# B&R Automation Studio project CombinedLinenCleanA6 (part 3)

#### 6_sdc1.var
```iecst
VAR RETAIN
	STEP : UINT;
	PLS : BOOL;
	LASTSTEP : UINT;
	SteadyUp : BOOL;
	CloserUpET : TIME;
	SteadysDown : BOOL;
	SteadysDownET : TIME;
	LoadDropped : BOOL;
END_VAR
VAR
	SteadyUpET : TIME;
	CloserDownET : TIME;
	SettledAtDischargerET : TIME;
	MinOpenET : TIME;
	SettledAtDischarger : BOOL;
	CloserDown : BOOL;
	MinOpen : BOOL;
	CloserUp : BOOL;
	SettledAtBuffer : BOOL;
	SettledAtBufferET : TIME;
	I_BagAtBuffer : BOOL;
	O_OpenStop : BOOL;
	O_OpenBag : BOOL;
	O_Steadys : BOOL;
	O_OpenBuffer : BOOL;
	O_Closer : BOOL;
	I_BagAtDischarger : BOOL;
	I_OpenBag : BOOL;
	I_LoadDropped : BOOL;
	TestDrop : BOOL;
	DischargerEnable : BOOL;
	TestDischarger : BOOL;
	Remainder : SINT;
	TimerAlarm : TON_10ms;
	WgtRound : UINT;
	a : BOOL;
	I_BagEmpty : BOOL;
	MySeq : USINT;
	O_BagReady : BOOL;
	O_JoinCDC4 : BOOL;
END_VAR
```

#### 6_sdc1Cyclic.ab
```automation-basic
PROGRAM _CYCLIC
	(* cyclic program *)

;Sequence 6 - Discharger 1 D[906]
a

;-----------------------------------------
;Revision 1.00 19/12/2005 D.J. First Issue
;-----------------------------------------

DischargerEnable 		= ((D[24] > 0) AND NOT Std.HaltSys)
MySeq                       = 9

//I_BagAtBuffer			  = X[3].X08
I_BagAtDischarger = X[3].X11
//I_SafetyRunning       = X[8].X15

I_OpenBag				= Enable.CDC4Open OR TestDrop           ;X[23].X01
//I_LoadDropped			= X[7].X13 OR TestDischarger  ;X[23].X02
//I_BagEmpty              = X[2].X13

O_Steadys				= FALSE ;Y[6].Y01
O_OpenBuffer 			= FALSE ;Y[6].Y02
O_OpenBag				= FALSE ;Y[6].Y03
O_OpenStop				= FALSE ;Y[6].Y04
O_Closer				= FALSE ;Y[6].Y05
O_BagReady          = FALSE
O_JoinCDC4           = FALSE
Request.CDC[4] 	     = FALSE

;Alarm
Alarm[MySeq].Name 			= 0 ;Clear sequence alarm name
Alarm[MySeq].Bag 			= 45
Alarm[MySeq].Beacon			= TRUE
Alarm[MySeq].Extra			= 0
Alarm[MySeq].Time			= 3000

;Setup Sequence
STEP = D[900+MySeq]
;Setup Pulse contact
PLS = (STEP <> LASTSTEP)
LASTSTEP = STEP

;Step 0 - Disabled
IF (STEP = 0) THEN
	;Disabled
ENDIF

;Check Status - Bag settled at buffer, no bag at discharger, bag at buffer on screen and no bag at discharger on the screen
TON_10ms(I_BagAtBuffer,300,SettledAtBuffer,SettledAtBufferET)
IF (STEP = 1) THEN
	IF DischargerEnable AND   NOT I_BagAtDischarger AND (Bag[45].Cat = 0) THEN
		D[900+MySeq] = 2
	ENDIF
	IF (Bag[45].Cat > 0) THEN
		Alarm[MySeq].Name = almBagDataError
	ELSE IF I_BagAtDischarger THEN
		Alarm[MySeq].Name = almSwitchFault
	ENDIF
ENDIF

;Wait for bag in discharger
IF (STEP = 2) THEN
	Request.CDC[4] 	= TRUE
;	IF (Bag[44].Cat = 0) AND (Bag[11].Cat>0) THEN
;		Bag[44] = Bag[11]
;		Bag[11]   = Bag[0]
;	ENDIF
	IF I_BagAtDischarger THEN
		D[900+MySeq] = 3
	ENDIF
	Alarm[7].Name = almBagNotArrived
ENDIF

;Let bag settle in discharger
TON_10ms(((STEP = 3) AND I_BagAtDischarger),1000,SettledAtDischarger,SettledAtDischargerET)
IF (STEP = 3) THEN
;	IF (Bag[228].Cat = 0) AND (Bag[227].Cat > 0) THEN
;		Bag[228] = Bag[227]
;		Bag[227] = Bag[0]
;	ENDIF
	IF SettledAtDischarger THEN
		D[900+MySeq] = 4
	ENDIF
	Alarm[MySeq].Name = almBagNotSettled
ENDIF

;Allow steadys to move down
TON_10ms((STEP = 4),400,SteadysDown,SteadysDownET)
IF (STEP = 4) THEN
	IF SteadysDown AND (Bag[45].Cat <> Std.MaxCats)  THEN
		D[900+MySeq] = 5
	ENDIF
	IF (Bag[45].Cat = Std.MaxCats) AND SteadysDown THEN
		D[900+MySeq] = 8
	ENDIF
ENDIF

;Steady cylinders on from steps 4 - 9
O_Steadys = ((STEP >= 4) AND (STEP <= 9))

;Bag opener on from step 5 - 8
O_OpenBag = ((STEP >= 6) AND (STEP <= 8))

;Wash Codes
;IF (STEP = 4) OR (STEP = 5) THEN
;
;;round up weight to give to wash machine
;	Remainder = SINT(Bag[228].Wgt MOD 10)
;	IF (Remainder > 4) THEN
;		WgtRound = (Bag[228].Wgt + 10)
;	ELSE
;		WgtRound = Bag[228].Wgt
;	ENDIF
;
;
;;Codes to CBW
;	CAN[1].Category = Bag[228].Cat
;	CAN[1].Customer = Bag[228].Cus
;	CAN[1].Weight   = (WgtRound / 10)
;ELSE
;	CAN[1].Category = 0
;	CAN[1].Customer = 0
;	CAN[1].Weight   = 0
;ENDIF

;Bag Ready to Washing Machine
IF (STEP = 5) THEN
	O_BagReady = TRUE
	O_Closer        = TRUE  ;  ????????????????????????
	IF I_OpenBag OR TestDischarger THEN
		D[900+MySeq] = 6
	ENDIF

ENDIF

;Open Bag Until LoadDropped recieved and has been open for 6 seconds
TON_10ms((STEP = 6),600,MinOpen,MinOpenET) ;ET means Elapsed Time
IF (STEP = 6) THEN
	IF  I_OpenBag THEN
		LoadDropped = TRUE
	ENDIF
	IF (NOT I_OpenBag AND MinOpen) THEN
		D[900+MySeq] = 7
	ENDIF
	Alarm[MySeq].Name = almLoadNotDropped
	ELSE
	LoadDropped = FALSE
ENDIF

;Change display to empty bag
IF (STEP = 7) THEN
	O_BagReady = Std.Clock500ms
	IF (D[927]>3) THEN
		LoadDropped = TRUE
	ENDIF
	IF (LoadDropped  OR TestDrop) THEN ;AND I_BagEmpty) OR TestDrop) THEN
		Bag[45].Cat 	= Std.MaxCats
		D[900+MySeq] 			= 8
	ENDIF
	Alarm[MySeq].Name = almGeneralSequence
	ELSE
	LoadDropped = FALSE
ENDIF

;Close bag
TON_10ms((STEP = 8),700,CloserDown,CloserDownET)
IF (STEP = 8) THEN
	O_Closer = TRUE
	IF CloserDown THEN
		D[900+MySeq] = 9
	ENDIF
ENDIF

;Allow closer to go back up
TON_10ms((STEP = 9),700,CloserUp,CloserUpET)
IF (STEP = 9) THEN
	IF CloserUp THEN
		D[900+MySeq] = 10
	ENDIF
ENDIF

;Allow steadys to go up
TON_10ms((STEP = 10),400,SteadyUp,SteadyUpET)
IF (STEP = 10) THEN
	IF SteadyUp THEN
		D[900+MySeq] = 11
	ENDIF
ENDIF

;Check for space on empty bag buffer
IF (STEP = 11) THEN
 	Request.CDC4Empty = TRUE
	IF Enable.CDC4Empty  THEN
		D[900+MySeq] = 12
	ENDIF
	ELSE
		Request.CDC4Empty = FALSE
ENDIF

;Open buffer stop - unitl bag out
IF (STEP = 12) THEN
	O_OpenStop = TRUE
	O_JoinCDC4 = TRUE
	IF PLS THEN
		Bag[42].Cat = 99
	ENDIF
	Bag[45].Cat = 0
	Bag[45].Cus = 0
	Bag[45].Wgt = 0
	IF NOT Enable.CDC4Empty AND NOT I_BagAtDischarger THEN
		D[900+MySeq] = 1
	ENDIF
	Alarm[MySeq].Name = almBagNotReleased
ENDIF

;Alarms
TimerAlarm.IN 	= NOT PLS AND (Alarm[MySeq].Name > 0)
TimerAlarm.PT 	= Alarm[MySeq].Time
TimerAlarm FUB TON_10ms()
Alarm[MySeq].On 	= TimerAlarm.Q
Alarm[MySeq].ET 	= TimerAlarm.ET

;Outputs

//Y[3].Y10 = O_OpenBuffer
Y[3].Y16 = O_Steadys
Y[4].Y01 = O_OpenBag
Y[4].Y02 = O_OpenStop
Y[4].Y03 = O_Closer
Y[7].Y01= O_JoinCDC4
END_PROGRAM
```

### Program Logical/Sequences/10ms/10_sdc5 (IEC, version 1.00.0) - * SDC1 Machine 1 BCD/CAN

#### 6_sdc1Cyclic.ab
```automation-basic
PROGRAM _CYCLIC
	(* cyclic program *)

;Sequence 6 - Discharger 1 D[906]
a

;-----------------------------------------
;Revision 1.00 19/12/2005 D.J. First Issue
;-----------------------------------------

DischargerEnable 		= ((D[25] > 0) AND NOT Std.HaltSys)
MySeq                       = 10

I_BagAtBuffer			  = X[3].X15
I_BagAtDischarger = X[3].X14
//I_SafetyRunning       = X[8].X15

I_OpenBag				= X[4].X01 OR TestDrop           ;X[23].X01
//I_LoadDropped			= X[7].X13 OR TestDischarger  ;X[23].X02
//I_BagEmpty              = X[2].X13

O_Steadys				= FALSE ;Y[6].Y01
O_OpenBuffer 			= FALSE ;Y[6].Y02
O_OpenBag				= FALSE ;Y[6].Y03
O_OpenStop				= FALSE ;Y[6].Y04
O_Closer				= FALSE ;Y[6].Y05
O_BagReady          = FALSE
Request.CDC[6]     = FALSE

;Alarm
Alarm[MySeq].Name 			= 0 ;Clear sequence alarm name
Alarm[MySeq].Bag 			= 46
Alarm[MySeq].Beacon			= TRUE
Alarm[MySeq].Extra			= 0
Alarm[MySeq].Time			= 3000

;Setup Sequence
STEP = D[900+MySeq]
;Setup Pulse contact
PLS = (STEP <> LASTSTEP)
LASTSTEP = STEP

;Step 0 - Disabled
IF (STEP = 0) THEN
	;Disabled
ENDIF

;Check Status - Bag settled at buffer, no bag at discharger, bag at buffer on screen and no bag at discharger on the screen
TON_10ms(I_BagAtBuffer,300,SettledAtBuffer,SettledAtBufferET)
IF (STEP = 1) THEN
	IF DischargerEnable AND SettledAtBuffer AND  NOT I_BagAtDischarger AND (Bag[46].Cat = 0) AND (Bag[26].Cat > 0)THEN
		D[900+MySeq] = 2
	ENDIF
	IF (Bag[46].Cat > 0) THEN
		Alarm[MySeq].Name = almBagDataError
	ELSE IF I_BagAtDischarger THEN
		Alarm[MySeq].Name = almSwitchFault
	ENDIF
ENDIF

;Wait for bag in discharger
IF (STEP = 2) THEN
	O_OpenBuffer 	= TRUE

	IF I_BagAtDischarger THEN
		D[900+MySeq] = 3
	ENDIF
	Alarm[7].Name = almBagNotArrived
ENDIF

;Let bag settle in discharger
TON_10ms(((STEP = 3) AND I_BagAtDischarger),1000,SettledAtDischarger,SettledAtDischargerET)
IF (STEP = 3) THEN
	IF (Bag[46].Cat = 0) AND (Bag[26].Cat>0) THEN
		Bag[46] = Bag[26]
		Bag[26]   = Bag[0]
	ENDIF
	IF SettledAtDischarger THEN
		D[900+MySeq] = 4
	ENDIF
	Alarm[MySeq].Name = almBagNotSettled
ENDIF

;Allow steadys to move down
TON_10ms((STEP = 4),400,SteadysDown,SteadysDownET)
IF (STEP = 4) THEN
	IF SteadysDown AND (Bag[46].Cat <> Std.MaxCats)  THEN
		D[900+MySeq] = 5
	ENDIF
	IF (Bag[46].Cat = Std.MaxCats) AND SteadysDown THEN
		D[900+MySeq] = 8
	ENDIF
ENDIF

;Steady cylinders on from steps 4 - 9
O_Steadys = ((STEP >= 4) AND (STEP <= 9))

;Bag opener on from step 5 - 8
O_OpenBag = ((STEP >= 6) AND (STEP <= 8))

;Wash Codes
;IF (STEP = 4) OR (STEP = 5) THEN
;
;;round up weight to give to wash machine
;	Remainder = SINT(Bag[228].Wgt MOD 10)
;	IF (Remainder > 4) THEN
;		WgtRound = (Bag[228].Wgt + 10)
;	ELSE
;		WgtRound = Bag[228].Wgt
;	ENDIF
;
;
;;Codes to CBW
;	CAN[1].Category = Bag[228].Cat
;	CAN[1].Customer = Bag[228].Cus
;	CAN[1].Weight   = (WgtRound / 10)
;ELSE
;	CAN[1].Category = 0
;	CAN[1].Customer = 0
;	CAN[1].Weight   = 0
;ENDIF

;Bag Ready to Washing Machine
IF (STEP = 5) THEN
	O_BagReady = TRUE
	O_Closer        = TRUE
	IF I_OpenBag OR TestDischarger THEN
		D[900+MySeq] = 6
	ENDIF

ENDIF

;Open Bag Until LoadDropped recieved and has been open for 6 seconds
TON_10ms((STEP = 6),600,MinOpen,MinOpenET) ;ET means Elapsed Time
IF (STEP = 6) THEN
	IF I_OpenBag THEN
		LoadDropped = TRUE
	ENDIF
	IF (NOT I_OpenBag AND MinOpen) THEN
		D[900+MySeq] = 7
	ENDIF
	Alarm[MySeq].Name = almLoadNotDropped
	ELSE
	LoadDropped = FALSE
ENDIF

;Change display to empty bag
IF (STEP = 7) THEN
	O_BagReady = TRUE
	IF I_OpenBag THEN
		LoadDropped = TRUE
	ENDIF
	IF (LoadDropped  OR TestDrop) THEN ;AND I_BagEmpty) OR TestDrop) THEN
		Bag[46].Cat 	= Std.MaxCats
		D[900+MySeq] 			= 8
	ENDIF
	Alarm[MySeq].Name = almGeneralSequence
	ELSE
	LoadDropped = FALSE
ENDIF

;Close bag
TON_10ms((STEP = 8),700,CloserDown,CloserDownET)
IF (STEP = 8) THEN
	O_Closer = TRUE
	IF CloserDown THEN
		D[900+MySeq] = 9
	ENDIF
ENDIF

;Allow closer to go back up
TON_10ms((STEP = 9),700,CloserUp,CloserUpET)
IF (STEP = 9) THEN
	IF CloserUp THEN
		D[900+MySeq] = 10
	ENDIF
ENDIF

;Allow steadys to go up
TON_10ms((STEP = 10),400,SteadyUp,SteadyUpET)
IF (STEP = 10) THEN
	IF SteadyUp THEN
		D[900+MySeq] = 11
	ENDIF
ENDIF

;Check for space on empty bag buffer
IF (STEP = 11) THEN
 	Request.CDC[5] = TRUE
	IF Enable.CDC[5]  THEN
		D[900+MySeq] = 12
	ENDIF
	ELSE
		Request.CDC[5] = FALSE
ENDIF

;Open buffer stop - unitl bag out
IF (STEP = 12) THEN
	O_OpenStop = TRUE
	IF PLS THEN
		;C[14] = 0
	ENDIF
	Bag[46].Cat = 0
	Bag[46].Cus = 0
	Bag[46].Wgt = 0
	IF NOT Enable.CDC[5]  THEN
		D[900+MySeq] = 1
	ENDIF
	Alarm[MySeq].Name = almBagNotReleased
ENDIF

;Alarms
TimerAlarm.IN 	= NOT PLS AND (Alarm[MySeq].Name > 0)
TimerAlarm.PT 	= Alarm[MySeq].Time
TimerAlarm FUB TON_10ms()
Alarm[MySeq].On 	= TimerAlarm.Q
Alarm[MySeq].ET 	= TimerAlarm.ET

;Outputs

Y[4].Y06 = O_OpenBuffer
Y[4].Y07 = O_Steadys
Y[4].Y08 = O_OpenBag
Y[4].Y09 = O_OpenStop
Y[4].Y10 = O_Closer

END_PROGRAM
```

#### 6_sdc1.var
```iecst
VAR RETAIN
	STEP : UINT;
	PLS : BOOL;
	LASTSTEP : UINT;
	SteadyUp : BOOL;
	CloserUpET : TIME;
	SteadysDown : BOOL;
	SteadysDownET : TIME;
	LoadDropped : BOOL;
END_VAR
VAR
	SteadyUpET : TIME;
	CloserDownET : TIME;
	SettledAtDischargerET : TIME;
	MinOpenET : TIME;
	SettledAtDischarger : BOOL;
	CloserDown : BOOL;
	MinOpen : BOOL;
	CloserUp : BOOL;
	SettledAtBuffer : BOOL;
	SettledAtBufferET : TIME;
	I_BagAtBuffer : BOOL;
	O_OpenStop : BOOL;
	O_OpenBag : BOOL;
	O_Steadys : BOOL;
	O_OpenBuffer : BOOL;
	O_Closer : BOOL;
	I_BagAtDischarger : BOOL;
	I_OpenBag : BOOL;
	I_LoadDropped : BOOL;
	TestDrop : BOOL;
	DischargerEnable : BOOL;
	TestDischarger : BOOL;
	Remainder : SINT;
	TimerAlarm : TON_10ms;
	WgtRound : UINT;
	a : BOOL;
	I_BagEmpty : BOOL;
	MySeq : USINT;
	O_BagReady : BOOL;
END_VAR
```

### Program Logical/Sequences/10ms/11_sdc6 (IEC) - * SDC1 Machine 1 BCD/CAN

#### 6_sdc1Cyclic.ab
```automation-basic
PROGRAM _CYCLIC
	(* cyclic program *)

;Sequence 6 - Discharger 1 D[906]
a

;-----------------------------------------
;Revision 1.00 19/12/2005 D.J. First Issue
;-----------------------------------------

DischargerEnable 		= ((D[26] > 0) AND NOT Std.HaltSys)
MySeq                       = 11

I_BagAtBuffer			  = X[6].X08
I_BagAtDischarger = X[4].X02
//I_SafetyRunning       = X[8].X15

I_OpenBag				= X[4].X04 OR TestDrop           ;X[23].X01
//I_LoadDropped			= X[7].X13 OR TestDischarger  ;X[23].X02
//I_BagEmpty              = X[2].X13

O_Steadys				= FALSE ;Y[6].Y01
O_OpenBuffer 			= FALSE ;Y[6].Y02
O_OpenBag				= FALSE ;Y[6].Y03
O_OpenStop				= FALSE ;Y[6].Y04
O_Closer				= FALSE ;Y[6].Y05
O_BagReady          = FALSE

;Alarm
Alarm[MySeq].Name 			= 0 ;Clear sequence alarm name
Alarm[MySeq].Bag 			= 47
Alarm[MySeq].Beacon			= TRUE
Alarm[MySeq].Extra			= 0
Alarm[MySeq].Time			= 3000

;Setup Sequence
STEP = D[900+MySeq]
;Setup Pulse contact
PLS = (STEP <> LASTSTEP)
LASTSTEP = STEP

;Step 0 - Disabled
IF (STEP = 0) THEN
	;Disabled
ENDIF

;Check Status - Bag settled at buffer, no bag at discharger, bag at buffer on screen and no bag at discharger on the screen
TON_10ms(I_BagAtBuffer,300,SettledAtBuffer,SettledAtBufferET)
IF (STEP = 1) THEN
	IF DischargerEnable AND SettledAtBuffer AND  NOT I_BagAtDischarger AND (Bag[47].Cat = 0) AND (Bag[21].Cat > 0)THEN
		D[900+MySeq] = 2
	ENDIF
	IF (Bag[47].Cat > 0) THEN
		Alarm[MySeq].Name = almBagDataError
	ELSE IF I_BagAtDischarger THEN
		Alarm[MySeq].Name = almSwitchFault
	ENDIF
ENDIF

;Wait for bag in discharger
IF (STEP = 2) THEN
	O_OpenBuffer 	= TRUE

	IF I_BagAtDischarger THEN
		D[900+MySeq] = 3
	ENDIF
	Alarm[7].Name = almBagNotArrived
ENDIF

;Let bag settle in discharger
TON_10ms(((STEP = 3) AND I_BagAtDischarger),1000,SettledAtDischarger,SettledAtDischargerET)
IF (STEP = 3) THEN
	IF (Bag[47].Cat = 0) AND (Bag[21].Cat>0) THEN
		Bag[47] = Bag[21]
		Bag[21]   = Bag[0]
	ENDIF
	IF SettledAtDischarger THEN
		D[900+MySeq] = 4
	ENDIF
	Alarm[MySeq].Name = almBagNotSettled
ENDIF

;Allow steadys to move down
TON_10ms((STEP = 4),400,SteadysDown,SteadysDownET)
IF (STEP = 4) THEN
	IF SteadysDown AND (Bag[47].Cat <> Std.MaxCats)  THEN
		D[900+MySeq] = 5
	ENDIF
	IF (Bag[47].Cat = Std.MaxCats) AND SteadysDown THEN
		D[900+MySeq] = 8
	ENDIF
ENDIF

;Steady cylinders on from steps 4 - 9
O_Steadys = ((STEP >= 4) AND (STEP <= 9))

;Bag opener on from step 5 - 8
O_OpenBag = ((STEP >= 6) AND (STEP <= 8))

;Wash Codes
;IF (STEP = 4) OR (STEP = 5) THEN
;
;;round up weight to give to wash machine
;	Remainder = SINT(Bag[228].Wgt MOD 10)
;	IF (Remainder > 4) THEN
;		WgtRound = (Bag[228].Wgt + 10)
;	ELSE
;		WgtRound = Bag[228].Wgt
;	ENDIF
;
;
;;Codes to CBW
;	CAN[1].Category = Bag[228].Cat
;	CAN[1].Customer = Bag[228].Cus
;	CAN[1].Weight   = (WgtRound / 10)
;ELSE
;	CAN[1].Category = 0
;	CAN[1].Customer = 0
;	CAN[1].Weight   = 0
;ENDIF

;Bag Ready to Washing Machine
IF (STEP = 5) THEN
	O_BagReady = TRUE
	O_Closer        = TRUE
	IF I_OpenBag OR TestDischarger THEN
		D[900+MySeq] = 6
	ENDIF

ENDIF

;Open Bag Until LoadDropped recieved and has been open for 6 seconds
TON_10ms((STEP = 6),600,MinOpen,MinOpenET) ;ET means Elapsed Time
IF (STEP = 6) THEN
	IF I_OpenBag THEN
//		LoadDropped = TRUE
	ENDIF
	IF (NOT I_OpenBag AND MinOpen) THEN
		D[900+MySeq] = 7
	ENDIF
;	Alarm[MySeq].Name = almLoadNotDropped
	ELSE
//	LoadDropped = FALSE
ENDIF

;Change display to empty bag
IF (STEP = 7) THEN
	O_BagReady = TRUE
	IF I_OpenBag THEN
		LoadDropped = TRUE
	ENDIF
	IF (LoadDropped  OR TestDrop) THEN ;AND I_BagEmpty) OR TestDrop) THEN
		Bag[47].Cat 	= Std.MaxCats
		D[900+MySeq] 			= 8
	ENDIF
	;Alarm[MySeq].Name = almGeneralSequence
	ELSE
	LoadDropped = FALSE
ENDIF

;Close bag
TON_10ms((STEP = 8),700,CloserDown,CloserDownET)
IF (STEP = 8) THEN
	O_Closer = TRUE
	IF CloserDown THEN
		D[900+MySeq] = 9
	ENDIF
ENDIF

;Allow closer to go back up
TON_10ms((STEP = 9),700,CloserUp,CloserUpET)
IF (STEP = 9) THEN
	IF CloserUp THEN
		D[900+MySeq] = 10
	ENDIF
ENDIF

;Allow steadys to go up
TON_10ms((STEP = 10),400,SteadyUp,SteadyUpET)
IF (STEP = 10) THEN
	IF SteadyUp THEN
		D[900+MySeq] = 11
	ENDIF
ENDIF

;Check for space on empty bag buffer
IF (STEP = 11) THEN
 	Request.CDC[6] = TRUE
	IF Enable.CDC[6]  THEN
		D[900+MySeq] = 12
	ENDIF
	ELSE
		Request.CDC[6] = FALSE
ENDIF

;Open buffer stop - unitl bag out
IF (STEP = 12) THEN
	O_OpenStop = TRUE
	IF PLS THEN
		;C[14] = 0
	ENDIF
	Bag[47].Cat = 0
	Bag[47].Cus = 0
	Bag[47].Wgt = 0
	IF NOT Enable.CDC[6]  THEN
		D[900+MySeq] = 1
	ENDIF
	Alarm[MySeq].Name = almBagNotReleased
ENDIF

;Alarms
TimerAlarm.IN 	= NOT PLS AND (Alarm[MySeq].Name > 0)
TimerAlarm.PT 	= Alarm[MySeq].Time
TimerAlarm FUB TON_10ms()
Alarm[MySeq].On 	= TimerAlarm.Q
Alarm[MySeq].ET 	= TimerAlarm.ET

;Outputs

Y[4].Y16 = O_BagReady
Y[8].Y16 = O_OpenBuffer
Y[4].Y12 = O_Steadys
Y[4].Y13 = O_OpenBag
Y[4].Y14 = O_OpenStop
Y[4].Y15 = O_Closer

END_PROGRAM
```

### Program Logical/Sequences/10ms/12_ebag (IEC) - *PUP1 Unloading point

#### pup.var
```iecst
VAR RETAIN
	LASTSTEP : UINT;
	PLS : BOOL;
	STEP : UINT;
END_VAR
VAR
	TimerAlarm : TON_10ms;
	mySeq : UINT;
	myIO : UINT;
	I_ReleasePB : BOOL;
	I_UnloadingPointOn : BOOL;
	I_TrolleyReleased : BOOL;
	I_BagAtBuffer : BOOL;
	I_BagReleasedBuffer : BOOL;
	myBag : UINT;
	O_Lamp : BOOL;
	O_OpenBuffer : BOOL;
	O_Release : BOOL;
	myPup : UINT;
	SettledBuffer : BOOL;
	SettledBufferET : UDINT;
	myBufferBag : UINT;
	BagReleased : BOOL;
	myZone : INT;
	I_BagInSep : BOOL;
	SettledInSep : BOOL;
	SettledInSepET : UDINT;
	O_SelectCDC3 : BOOL;
	O_SelectCIC3 : BOOL;
END_VAR
```

#### pup.ab
```automation-basic
;--------------------------------------------
;Sequence 0 - XXX0  D[900 + mySeq]
;--------------------------------------------

PROGRAM _INIT
(* init program *)
END_PROGRAM

PROGRAM _CYCLIC

;Inputs
mySeq				= 12	;Sequence number
//myIO				= 345
//myBu/fferBag			= 950
//myBa/g				= 987
//myPup				= 1
//myZone				= 0

I_BagAtBuffer		= X[myIO].X01
I_BagInSep			= X[myIO].X02
I_UnloadingPointOn	= X[myIO].X03
I_ReleasePB			= X[myIO].X04
I_TrolleyReleased	= X[myIO].X08 ; Also Line full

Enable.CDC[3]  = FALSE
Enable.CIC[3]    = FALSE

//PUP[myPup].WorkingLamp = FALSE
O_SelectCIC3        = FALSE
O_SelectCDC3       = FALSE

Alarm[mySeq].Name 	= 0
Alarm[mySeq].Bag	= myBag
Alarm[mySeq].Beacon	= TRUE
Alarm[mySeq].Extra	= 0
Alarm[mySeq].Time	= 3000

;Setup Sequence
STEP = D[900 + mySeq]
;Setup Pulse contact
PLS = (STEP <> LASTSTEP)
LASTSTEP = STEP

;Sequence
IF (STEP = 0) THEN
	;Disabled
ENDIF

;Step 1 Wiat for bag at buffer.
TON_10ms(I_BagAtBuffer,75,SettledBuffer,SettledBufferET)
IF (STEP = 1) THEN
	IF Line[9].Clear THEN
		D[900 + mySeq] = 2
	ENDIF
	//	Alarm[mySeq].Name = almBagDataError

ENDIF

;Step 2 Release bag from Buffer
//TON_10ms(I_BagInSep,150,SettledInSep,SettledInSepET)
IF (STEP = 2) THEN
	IF Request.CDC[3] THEN
		C[9] = 0
		D[900 + mySeq] = 3
	ELSE IF Request.CIC[3] THEN
		C[9] = 0
		D[900 + mySeq] = 4
	ENDIF
	//	Alarm[mySeq].Bag = myBufferBag
	//	Alarm[mySeq].Name = almBagNotReleased

ENDIF

;Step 3 wait for pushbutton to request release of trolley
IF (STEP = 3) THEN
	O_SelectCDC3 = TRUE
	Enable.CDC[3] = TRUE
	IF Line[9].Trip THEN
		D[900 + mySeq] = 1
	ENDIF
		Alarm[mySeq].Name = almBagNotArrived
ENDIF

;STEP 4 Check for space in empty trolley buffer.
IF (STEP = 4) THEN
	O_SelectCIC3 = TRUE
	Enable.CIC[3]  = TRUE
	IF Line[9].Trip THEN
		D[900 + mySeq] = 1
	ENDIF
		Alarm[mySeq].Name = almBagNotArrived
ENDIF

;-----------------------------------
;PLC Outputs - adjust to suit system
;-----------------------------------

Y[6].Y10 = O_SelectCIC3
Y[6].Y09 = O_SelectCDC3

;Alarms
TimerAlarm.IN 		= NOT PLS AND (Alarm[mySeq].Name > 0)
TimerAlarm.PT 		= Alarm[mySeq].Time
TimerAlarm FUB TON_10ms()
Alarm[mySeq].On 	= TimerAlarm.Q
Alarm[mySeq].ET 	= TimerAlarm.ET
//Alarm[mySeq].Zone 	= myZone
END_PROGRAM
```

### Program Logical/Sequences/10ms/13_fb_eb (IEC) - *PUP5 Unloading point

#### pup.var
```iecst
VAR RETAIN
	LASTSTEP : UINT;
	PLS : BOOL;
	STEP : UINT;
END_VAR
VAR
	TimerAlarm : TON_10ms;
	mySeq : UINT;
	myIO : UINT;
	I_ReleasePB : BOOL;
	I_UnloadingPointOn : BOOL;
	I_TrolleyReleased : BOOL;
	myBag : UINT;
	O_Lamp : BOOL;
	O_OpenBuffer : BOOL;
	O_Release : BOOL;
	myPup : UINT;
	SettledBuffer : BOOL;
	SettledBufferET : UDINT;
	PUPValid : BOOL;
	myZone : INT;
	I_BagAtEmpty : BOOL;
	I_BagAtLine1 : BOOL;
	I_BagAtLine2 : BOOL;
	I_CDC1PB : BOOL;
	I_CDC1SelectLine1 : BOOL;
	I_CDC1SelectLine4 : BOOL;
	I_CDC4PB : BOOL;
	I_CDC4SelectLine1 : BOOL;
	I_CDC4SelectLine4 : BOOL;
	O_ResetPoints : BOOL;
	O_OpenEmpty : BOOL;
	O_OpenLine1 : BOOL;
	O_OpenLine2 : BOOL;
	O_SelectCDC1 : BOOL;
	O_SelectCDC4 : BOOL;
	O_JoinCDC4 : BOOL;
	O_JoinCDC1 : BOOL;
	PointsReset : BOOL;
	PointsResetET : UDINT;
	SettledAtEmpty : BOOL;
	SettledAtEmptyET : UDINT;
	Alt : USINT;
	AlternateBetweenLine1And4 : BOOL;
	SettledAtLine1 : BOOL;
	SettledAtLine2 : BOOL;
	E : BOOL;
	SettledAtCDC1ET : UDINT;
	SettledAtCDC4ET : UDINT;
END_VAR
```

#### pup.ab
```automation-basic
;--------------------------------------------
;Sequence 0 - XXX0  D[900 + mySeq]
;--------------------------------------------

PROGRAM _INIT
(* init program *)
END_PROGRAM

PROGRAM _CYCLIC

;Inputs
mySeq				= 13	;Sequence number

I_BagAtEmpty		= X[6].X12
I_BagAtLine1		= X[6].X11
I_BagAtLine2		= X[6].X13

I_CDC1PB			= X[6].X15
I_CDC1SelectLine1	= X[8].X08
I_CDC1SelectLine4	= X[8].X09

I_CDC4PB			= X[6].X16
I_CDC4SelectLine1	= X[8].X05
I_CDC4SelectLine4	= X[8].X06

O_ResetPoints	= FALSE
O_OpenEmpty		= FALSE
O_OpenLine1		= FALSE
O_OpenLine2		= FALSE
O_SelectCDC1	= FALSE
O_SelectCDC4	= FALSE
O_JoinCDC4		= FALSE
O_JoinCDC1		= FALSE

Alarm[mySeq].Name 	= 0
Alarm[mySeq].Bag	= 1
Alarm[mySeq].Beacon	= TRUE
Alarm[mySeq].Extra	= 0
Alarm[mySeq].Time	= 3000

;Setup Sequence
STEP = D[900 + mySeq]
;Setup Pulse contact
PLS = (STEP <> LASTSTEP)
LASTSTEP = STEP

;Sequence
IF (STEP = 0) THEN
	;Disabled
ENDIF

TON_10ms((STEP = 1),300,PointsReset,PointsResetET)

;Reset Points
IF (STEP = 1) THEN
//	D[45] = 0
//	D[46] = 0
	O_ResetPoints = TRUE
	IF PointsReset THEN
	D[913] = 2
 	ENDIF
ENDIF

TON_10ms(I_BagAtEmpty,300,SettledAtEmpty,SettledAtEmptyET)
TON_10ms((I_BagAtLine1 AND (Bag[1].Cat  > 0)),300,SettledAtLine1 ,SettledAtCDC1ET)
TON_10ms((I_BagAtLine2 AND (Bag[16].Cat > 0)),300,SettledAtLine2 ,SettledAtCDC4ET)
IF (STEP = 2) THEN
	IF (Alt > 2) THEN
		Alt = 0
	ENDIF
	IF Request.CDC[4] AND NOT I_CDC4SelectLine1 AND NOT I_CDC4SelectLine4 THEN
		AlternateBetweenLine1And4 = TRUE
	ELSE
		AlternateBetweenLine1And4 = FALSE
	ENDIF

	IF 	AlternateBetweenLine1And4 THEN
		Alt = Alt + 1
	ENDIF
;	IF ((Bag[41].Cat= 0) AND Request.CIC[4] AND SettledAtLine1) THEN ;CDC1 Request For Bag From Line 1
	;	D[913] = 3
;	ELSE IF ((Bag[41].Cat= 0) AND Request.CDC[1] AND SettledAtLine2 AND I_CDC1PB AND I_CDC1SelectLine4) THEN ;CDC1 Request For Bag From Line 2
		;D[913] = 4
	 IF ((Bag[41].Cat = 0) AND Request.CDC[4] AND SettledAtLine1  AND (I_CDC4SelectLine1 OR AlternateBetweenLine1And4 AND (Alt = 1))) THEN ;CDC4 Request For Bag From Line 1
		D[913]	= 3
	ELSE IF ((Bag[41].Cat = 0) AND Request.CDC[4] AND SettledAtLine2  AND (I_CDC4SelectLine4 OR AlternateBetweenLine1And4 AND (Alt = 2))) THEN ;CDC4 Request For Bag From Line 2
		D[913]	= 4
	ELSE IF ((Bag[41].Cat = 0) AND Request.CIC[4] AND SettledAtEmpty AND NOT I_CDC4PB AND NOT I_CDC1PB AND NOT Request.CDC4Empty) THEN  ;No Full Bags To Send Or Empty Bags Needed
		Bag[41].Cat = 99
		D[913]	= 5
	ENDIF
ENDIF

;Line 1 Bag To CDC1
IF (STEP = 9) THEN
	O_OpenLine1 	= TRUE
	O_SelectCDC1	= TRUE
	O_JoinCDC1		= TRUE
	IF (Bag[1].Cat>0) AND (Bag[41].Cat=0) THEN
				Bag[41].Cat = 99
				Bag[1] = Bag[0]
	ENDIF
//	D[45]			= 1
//	D[46]			= 1
//	D[47] 			= 2
			Alarm[mySeq].Name = almBagNotArrived
	IF NOT Request.CDC[1] THEN
		IF (Bag[41].Cat>0) AND (Bag[42].Cat=0) THEN
				Bag[42] = Bag[41]
				Bag[41] = Bag[0]
			ENDIF
		D[913] = 1
	ENDIF
ENDIF

;Line 4 Bag To CDC1
IF (STEP = 8) THEN
	O_OpenLine2 	= TRUE
	O_SelectCDC1	= TRUE
	O_JoinCDC1		= TRUE
	IF (Bag[16].Cat>0) AND (Bag[41].Cat=0) THEN
				Bag[41] = Bag[16]
				Bag[16] = Bag[0]
			ENDIF
	D[45]			= 4
	D[46]			= 1
	D[47]			= 1
			Alarm[mySeq].Name = almBagNotArrived
	IF NOT Request.CIC[4] THEN
	//	BAGMOVE2(TRUE,mem_adr_E,41,42,BagSpacing)
		IF (Bag[41].Cat>0) AND (Bag[42].Cat=0) THEN
				Bag[42] = Bag[41]
				Bag[41] = Bag[0]
			ENDIF
		D[913] = 1
	ENDIF
ENDIF

;Line 1 Bag To CDC4
IF (STEP = 3) THEN
	O_OpenLine1 	= TRUE
	O_SelectCDC4	= TRUE
	;O_JoinCDC1		= TRUE
		IF (Bag[1].Cat>0) AND (Bag[41].Cat=0) THEN
				Bag[41] = Bag[1]
				Bag[1] = Bag[0]
			ENDIF
			Alarm[mySeq].Name = almBagNotArrived
	D[45]			= 1
	D[46]			= 4
//	E[204]			= 107			;Set dest to CDC1
	IF NOT Request.CDC[4] THEN
//		BAGMOVE2(TRUE,mem_adr_E,41,45,BagSpacing)
		IF (Bag[41].Cat>0) AND (Bag[45].Cat=0) THEN
				Bag[45] = Bag[41]
				Bag[41] = Bag[0]
			ENDIF
		D[913] = 1
	ENDIF
ENDIF

;Line 4 Bag To CDC4
IF (STEP = 4) THEN
	O_OpenLine2 	= TRUE
	O_SelectCDC4	= TRUE
	;O_JoinCDC1		= TRUE
		IF (Bag[16].Cat>0) AND (Bag[41].Cat=0) THEN
				Bag[41] = Bag[16]
				Bag[16] = Bag[0]
			ENDIF
//	BAGMOVE2(TRUE,mem_adr_E,16,41,BagSpacing)
//	D[45]			= 4
//	D[46]			= 4
//	E[204]			= 107			;Set dest to CDC1
	IF NOT Request.CDC[4] THEN
//		BAGMOVE2(TRUE,mem_adr_E,41,45,BagSpacing)
		IF (Bag[41].Cat>0) AND (Bag[45].Cat=0) THEN
				Bag[45] = Bag[41]
				Bag[41] = Bag[0]
			ENDIF
		D[913] = 1
	ENDIF
ENDIF

;Empty bags to CDC1
IF (STEP = 5) THEN
	O_OpenEmpty 	= TRUE
	O_SelectCDC1	= TRUE
	O_JoinCDC1		= TRUE
//	D[45]			= 2
//	D[46]			= 1
//	D[47]			= 1
//	E[200]			= Std.MaxCats 	;Set BIT to Empty
			Alarm[mySeq].Name = almBagNotArrived
	IF X[3].X01 THEN
//		BAGMOVE2(TRUE,mem_adr_E,41,42,BagSpacing)
		IF (Bag[41].Cat>0) AND (Bag[42].Cat=0) THEN
				Bag[42] = Bag[41]
				Bag[41] = Bag[0]
			ENDIF
		D[913] = 1
	ENDIF
ENDIF

IF ((STEP = 0) OR (STEP = 1) OR (STEP = 2)) THEN
	D[45] = 0
	D[46] = 0
	D[47] = 0
ENDIF

;-----------------------------------
;PLC Outputs - adjust to suit system
;-----------------------------------

Y[6].Y12 = O_ResetPoints
Y[6].Y16 = O_OpenEmpty
Y[6].Y11 = O_OpenLine1
Y[6].Y13 = O_OpenLine2
Y[6].Y15 = O_SelectCDC1
Y[6].Y14 = O_SelectCDC4
;Y701 = O_JoinCDC4
Y[7].Y02 = O_JoinCDC1

;Alarms
TimerAlarm.IN 		= NOT PLS AND (Alarm[mySeq].Name > 0)
TimerAlarm.PT 		= Alarm[mySeq].Time
TimerAlarm FUB TON_10ms()
Alarm[mySeq].On 	= TimerAlarm.Q
Alarm[mySeq].ET 	= TimerAlarm.ET
//Alarm[mySeq].Zone 	= myZone
END_PROGRAM
```

### Program Logical/Sequences/10ms/14_cvc2 (IEC, version 1.00.0) - * SVC1 Up from SLU1 & Loading

#### 8_svc1Cyclic.ab
```automation-basic
PROGRAM _CYCLIC
	(* cyclic program *)

;--------------------------------------------
;Sequence 8 - SVC1 Vertical conveyor 1 D[908]
;--------------------------------------------

;--------------------------------------------
;Sequence 52 - CVC1 Vertical conveyor 1 D[952]
;--------------------------------------------

;Inputs
I_CarriageAtTop			= X[4].X13
I_CarriageAtBottom		= X[4].X14
I_BagOnCarriage			= X[4].X15
I_BagAtBuffer1			= X[7].X04 AND (D[29]>0)
I_BagAtBuffer2			= X[7].X03 AND (D[19]>0)

O_MoveUp 				= FALSE
O_MoveDown 				= FALSE
O_OpenStop 				= FALSE
O_Select1				= FALSE
O_Select2				= FALSE

//Enable.LU[1]			= FALSE

Alarm[14].Name 				= 0
Alarm[14].Bag				= 10001
Alarm[14].Beacon			= TRUE
Alarm[14].Extra				= 0
Alarm[14].Time			  	= 5000

;Setup Sequence
STEP = D[914]
;Setup Pulse contact
PLS = (STEP <> LASTSTEP)
LASTSTEP = STEP

;Alarm
;TON_10ms(((NOT PLS) AND (STEP <> 2) AND (STEP <> 6)AND (STEP <> 10)AND (STEP <> 11)AND (STEP <> 14) AND (STEP <> 16)),3000,Alarm[52],AlarmET[52])

;Sequence
IF (STEP = 0) THEN
	;Disabled
ENDIF

;Move bag from LU to Carriage
IF (STEP = 1) THEN
O_MoveUp = (NOT I_CarriageAtTop AND NOT I_BagOnCarriage)
	IF I_CarriageAtTop THEN
		D[914] = 2
	ENDIF
ENDIF

TON_10ms(I_BagAtBuffer1,300,SettledAtBuffer1,SettledAtBuffer1ET)
TON_10ms(I_BagAtBuffer2,300,SettledAtBuffer2,SettledAtBuffer2ET)
IF (STEP = 2) THEN
	Alternator = Alternator + 1
	IF (Alternator > 3) THEN
		Alternator = 1
	ENDIF
	IF (SettledAtBuffer2) THEN
		D[48]	= 2
		D[914]	= 3
	ELSE IF ( SettledAtBuffer1) THEN
		D[48]	= 1
		D[914]	= 3
	ELSE IF ((Alternator = 3) AND SettledAtBuffer1) THEN
		;D[48]	= 1
		;D[914]	= 3
	ENDIF
ENDIF

;Bag moves to carriage
TON_10ms(I_BagOnCarriage,300,SettledOnCarriage,SettledOnCarriageET)
IF (STEP = 3) THEN
	O_Select1 = ((D[48] = 1) AND I_CarriageAtTop)
	O_Select2 = ((D[48] = 2) AND I_CarriageAtTop)
	IF I_BagOnCarriage THEN
		D[914] = 4
	ENDIF
ENDIF

;Clear route selection
IF (STEP <> 2) AND (STEP <> 3) THEN
	D[48] = 0
ENDIF

;Bag Settles on carriage
TON_10ms(I_BagOnCarriage,200,SettledOnCarriage,SettledOnCarriageET)
IF (STEP = 4) THEN
	IF SettledOnCarriage THEN
		D[914] = 5
	ENDIF
ENDIF

;Move carriage down to bottom
IF (STEP = 5) THEN
	O_MoveDown = (NOT I_CarriageAtBottom)
	IF I_CarriageAtBottom THEN
		D[914] = 6
	ENDIF
ENDIF

;Wait for loading unit to call the bag
IF (STEP = 6) THEN
	IF Enable.CVC[2] THEN
		D[914] = 7
	ENDIF
ENDIF

;Bag arrves at loading unit
IF (STEP = 7) THEN
	O_OpenStop = I_CarriageAtBottom
	IF NOT Enable.CVC[2] THEN
		D[914] = 1
	ENDIF
ENDIF

;High Speed Used For Up		= 50Hz
;Medium Speed Used For Down	= 50Hz

TON_10ms(O_MoveUp  ,700,HighSpeedUp,HighSpeedUpET) 		;Expected 16.94 seconds @ 591mm/sec
TON_10ms(O_MoveDown,700,HighSpeedDn,HighSpeedDnET) 		;Expected 16.94 seconds @ 591mm/sec
IF (STEP = 1) THEN
	Y[8].Y03 = (NOT HighSpeedUp) 							;High Speed
	Y[8].Y04 = FALSE										;Medium Speed
ELSE IF (STEP = 5) THEN
	Y[8].Y03 = FALSE										;High Speed
	Y[8].Y04 = (NOT HighSpeedDn)							;Medium Speed
ELSE
	Y[8].Y03 = FALSE
	Y[8].Y04 = FALSE
ENDIF

;PLC Outputs
;-----------
Y[9].Y05 = O_MoveUp
Y[9].Y06 = O_MoveDown
Y[9].Y07 = (O_MoveUp OR O_MoveDown)
Y[9].Y08 = O_OpenStop

Y[7].Y04 = O_Select1
Y[7].Y03 = O_Select2

END_PROGRAM
```

#### 8_svc1.var
```iecst
VAR
	I_CarrAtTop : BOOL;
	I_CarrAtBottom : BOOL;
END_VAR
VAR RETAIN
	STEP : UINT;
	PLS : BOOL;
END_VAR
VAR
	LASTSTEP : UINT;
	O_MoveCarrUp : BOOL;
	O_OpenCarrStop : BOOL;
	O_MoveCarrDown : BOOL;
	I_BagOnCarr : BOOL;
	O_OpenBuffer : BOOL;
	BagSettledOnCarr : BOOL;
	BagSettledOnCarrET : TIME;
	I_BagReleased : BOOL;
	TimerAlarm : TON_10ms;
	I_CarrAtMiddle : BOOL;
	I_CarrAtWeighing : BOOL;
	I_NoEmptyBag : BOOL;
	I_CollectEmpty : BOOL;
	I_UseAsLoading : BOOL;
	I_UpPushButton : BOOL;
	I_DownPushButton : BOOL;
	Dst : UINT;
	PButton : BOOL;
	SVCRaw : DINT;
	n : UINT;
	ValidCus : BOOL;
	ValidWgt : BOOL;
	O_AlarmLamp : BOOL;
	ValidCat : BOOL;
	Choice : ARRAY[0..4] OF UINT;
	PButtonET : TIME;
	Status : UINT;
	PastMiddleET : TIME;
	PastMiddle : BOOL;
	ValidDst : BOOL;
	I_CarrAtEmptyBagIn : BOOL;
	I_CarrAtEmptyBagOut : BOOL;
	I_BagAtBufferStopLLevel : BOOL;
	I_BagAtEmptyBufferStop : BOOL;
	O_OpenEmptyBufferStop : BOOL;
	O_OpenFullbufferStop : BOOL;
	MoveDownEmptyOut : BOOL;
	O_BufferStop : BOOL;
	AlarmET : UDINT;
	SettledEmptyBuffer : BOOL;
	SettledEmptyBufferET : UDINT;
	SettledOnCarr : BOOL;
	SettledOnCarrET : UDINT;
	EmptyBufferClear : BOOL;
	SettledBuffer : BOOL;
	SettledBufferET : UDINT;
	EmptyDownToEmptyIn : BOOL;
	EmptyDownToEmptyInET : UDINT;
	EmptyDownToEmptyOut : BOOL;
	EmptyDownToEmptyOutET : UDINT;
	EmptyDownToFullIn : BOOL;
	EmptyDownToFullInET : UDINT;
	UpToTop : BOOL;
	UpToTopET : UDINT;
	O_MoveDownEmptyOut : BOOL;
	ReleaseBrake : BOOL;
	MoveDownStep : BOOL;
	MoveUpStep : BOOL;
	HighSpeedTime : UINT;
	TONHighSpeed : TON_10ms;
	HighSpeedDone : BOOL;
	HighSpeedDoneET : TIME;
	O_Point1_4 : BOOL;
	O_Point5 : BOOL;
	StopDelay : BOOL;
	StopDelayET : UDINT;
	TONSteadys : TON_10ms;
	O_CarriageSteadys : BOOL;
	I_CarriageAtTop : BOOL;
	I_CarriageAtBottom : BOOL;
	I_BagOnCarriage : BOOL;
	I_BagAtBuffer1 : BOOL;
	I_BagAtBuffer2 : BOOL;
	O_MoveUp : BOOL;
	O_MoveDown : BOOL;
	O_OpenStop : BOOL;
	O_Select1 : BOOL;
	O_Select2 : BOOL;
	SettledAtBuffer1 : BOOL;
	SettledAtBuffer1ET : UDINT;
	SettledAtBuffer2 : BOOL;
	SettledAtBuffer2ET : UDINT;
	Alternator : USINT;
	SettledOnCarriage : BOOL;
	SettledOnCarriageET : UDINT;
	HighSpeedUp : BOOL;
	HighSpeedUpET : UDINT;
	HighSpeedDn : BOOL;
	HighSpeedDnET : UDINT;
END_VAR
```

### Program Logical/Sequences/10ms/15_cdc7 (IEC) - * SDC1 Machine 1 BCD/CAN

#### 6_sdc1Cyclic.ab
```automation-basic
PROGRAM _CYCLIC
	(* cyclic program *)

;Sequence 6 - Discharger 1 D[906]
a

;-----------------------------------------
;Revision 1.00 19/12/2005 D.J. First Issue
;-----------------------------------------

DischargerEnable 		= ((D[27] > 0) AND NOT Std.HaltSys)
MySeq                       = 15

I_BagAtBuffer			  = X[7].X01
I_BagAtDischarger = X[4].X05
//I_SafetyRunning       = X[8].X15

I_OpenBag				= Enable.CDC[7] OR TestDrop           ;X[23].X01
//I_LoadDropped			= X[7].X13 OR TestDischarger  ;X[23].X02
I_BagOut             = X[4].X06

O_Steadys				= FALSE ;Y[6].Y01
O_OpenBuffer 			= FALSE ;Y[6].Y02
O_OpenBag				= FALSE ;Y[6].Y03
O_OpenStop				= FALSE ;Y[6].Y04
O_Closer				= FALSE ;Y[6].Y05
O_BagReady          = FALSE

;Alarm
Alarm[MySeq].Name 			= 0 ;Clear sequence alarm name
Alarm[MySeq].Bag 			= 48
Alarm[MySeq].Beacon			= TRUE
Alarm[MySeq].Extra			= 0
Alarm[MySeq].Time			= 3000

;Setup Sequence
STEP = D[900+MySeq]
;Setup Pulse contact
PLS = (STEP <> LASTSTEP)
LASTSTEP = STEP

;Step 0 - Disabled
IF (STEP = 0) THEN
	;Disabled
ENDIF

;Check Status - Bag settled at buffer, no bag at discharger, bag at buffer on screen and no bag at discharger on the screen
TON_10ms(I_BagAtBuffer,300,SettledAtBuffer,SettledAtBufferET)
IF (STEP = 1) THEN
	IF DischargerEnable AND SettledAtBuffer AND  NOT I_BagAtDischarger AND (Bag[48].Cat = 0) AND (Bag[63].Cat > 0)THEN
		D[900+MySeq] = 2
	ENDIF
	IF (Bag[63].Cat > 0) THEN
		Alarm[MySeq].Name = almBagDataError
	ELSE IF I_BagAtDischarger THEN
		Alarm[MySeq].Name = almSwitchFault
	ENDIF
ENDIF

;Wait for bag in discharger
IF (STEP = 2) THEN
	O_OpenBuffer 	= TRUE

	IF I_BagAtDischarger THEN
		D[900+MySeq] = 3
	ENDIF
	Alarm[7].Name = almBagNotArrived
ENDIF

;Let bag settle in discharger
TON_10ms(((STEP = 3) AND I_BagAtDischarger),1000,SettledAtDischarger,SettledAtDischargerET)
IF (STEP = 3) THEN
	IF (Bag[48].Cat = 0) AND (Bag[63].Cat>0) THEN
		Bag[48] = Bag[63]
		Bag[63]   = Bag[0]
	ENDIF
	IF SettledAtDischarger THEN
		D[900+MySeq] = 4
	ENDIF
	Alarm[MySeq].Name = almBagNotSettled
ENDIF

;Allow steadys to move down
TON_10ms((STEP = 4),400,SteadysDown,SteadysDownET)
IF (STEP = 4) THEN
	IF SteadysDown AND (Bag[48].Cat <> Std.MaxCats)  THEN
		D[900+MySeq] = 5
	ENDIF
	IF (Bag[48].Cat = Std.MaxCats) AND SteadysDown THEN
		D[900+MySeq] = 8
	ENDIF
ENDIF

;Steady cylinders on from steps 4 - 9
O_Steadys = ((STEP >= 4) AND (STEP <= 9))

;Bag opener on from step 5 - 8
O_OpenBag = ((STEP >= 6) AND (STEP <= 8))

;Wash Codes
;IF (STEP = 4) OR (STEP = 5) THEN
;
;;round up weight to give to wash machine
;	Remainder = SINT(Bag[228].Wgt MOD 10)
;	IF (Remainder > 4) THEN
;		WgtRound = (Bag[228].Wgt + 10)
;	ELSE
;		WgtRound = Bag[228].Wgt
;	ENDIF
;
;
;;Codes to CBW
;	CAN[1].Category = Bag[228].Cat
;	CAN[1].Customer = Bag[228].Cus
;	CAN[1].Weight   = (WgtRound / 10)
;ELSE
;	CAN[1].Category = 0
;	CAN[1].Customer = 0
;	CAN[1].Weight   = 0
;ENDIF

;Bag Ready to Washing Machine
IF (STEP = 5) THEN
	O_BagReady = TRUE
	O_Closer        = TRUE
	IF I_OpenBag OR TestDischarger THEN
		D[900+MySeq] = 6
	ENDIF

ENDIF

;Open Bag Until LoadDropped recieved and has been open for 6 seconds
TON_10ms((STEP = 6),600,MinOpen,MinOpenET) ;ET means Elapsed Time
IF (STEP = 6) THEN
	IF (D[924]>3) THEN
		LoadDropped = TRUE
	ENDIF
	IF (NOT I_OpenBag AND MinOpen) THEN
		D[900+MySeq] = 7
	ENDIF
	Alarm[MySeq].Name = almLoadNotDropped
	ELSE
//	LoadDropped = FALSE
ENDIF

;Change display to empty bag
IF (STEP = 7) THEN

	IF (NOT I_OpenBag OR TestDrop) THEN ;AND I_BagEmpty) OR TestDrop) THEN
		Bag[48].Cat 	= Std.MaxCats
		D[900+MySeq] 			= 8
	ENDIF
	Alarm[MySeq].Name = almGeneralSequence
	ELSE
	LoadDropped = FALSE
ENDIF

;Close bag
TON_10ms((STEP = 8),700,CloserDown,CloserDownET)
IF (STEP = 8) THEN
	O_Closer = TRUE
	IF CloserDown THEN
		D[900+MySeq] = 9
	ENDIF
ENDIF

;Allow closer to go back up
TON_10ms((STEP = 9),700,CloserUp,CloserUpET)
IF (STEP = 9) THEN
	IF CloserUp THEN
		D[900+MySeq] = 10
	ENDIF
ENDIF

;Allow steadys to go up
TON_10ms((STEP = 10),400,SteadyUp,SteadyUpET)
IF (STEP = 10) THEN
	IF SteadyUp THEN
		D[900+MySeq] = 11
	ENDIF
ENDIF

;Check for space on empty bag buffer
IF (STEP = 11) THEN

ENDIF

;Open buffer stop - unitl bag out
IF (STEP = 12) THEN
	O_OpenStop = TRUE
	IF PLS THEN
		;C[14] = 0
	ENDIF
	Bag[48].Cat = 0
	Bag[48].Cus = 0
//	Bag[48.Wgt = 0
	IF I_BagOut   THEN
		D[900+MySeq] = 1
	ENDIF
	Alarm[MySeq].Name = almBagNotReleased
ENDIF

;Alarms
TimerAlarm.IN 	= NOT PLS AND (Alarm[MySeq].Name > 0)
TimerAlarm.PT 	= Alarm[MySeq].Time
TimerAlarm FUB TON_10ms()
Alarm[MySeq].On 	= TimerAlarm.Q
Alarm[MySeq].ET 	= TimerAlarm.ET

;Outputs

//Y[4].Y16 = O_BagReady
Y[2].Y15 = O_OpenBuffer
Y[5].Y01 = O_Steadys
Y[5].Y02 = O_OpenBag
Y[5].Y03 = O_OpenStop
Y[5].Y04 = O_Closer

END_PROGRAM
```

### Program Logical/Sequences/10ms/16_cic4 (IEC) - * SPC1 Empty bags up

#### 9_spc1.var
```iecst
VAR
	I_CarrAtTop : BOOL;
	I_CarrAtBottom : BOOL;
END_VAR
VAR RETAIN
	STEP : UINT;
END_VAR
VAR
	PLS : BOOL;
END_VAR
VAR RETAIN
	LASTSTEP : UINT;
END_VAR
VAR
	O_MoveCarrUp : BOOL;
	O_OpenCarrStop : BOOL;
	O_MoveCarrDown : BOOL;
	I_BagOnCarr : BOOL;
	O_OpenBuffer : BOOL;
	SettledBuffer : BOOL;
	SettledBufferET : TIME;
	I_BagAtBuffer : BOOL;
	BagSettledOnCarr : BOOL;
	BagSettledOnCarrET : TIME;
	I_BagReleased : BOOL;
	TimerAlarm : TON_10ms;
	I_BagAtLLBuff : BOOL;
	O_LLBuffOpen : BOOL;
	SettledBufferSDC2ET : TIME;
	SettledBufferSDC2 : BOOL;
	I_BagAtBufferSDC2 : BOOL;
	Alt : USINT;
	O_OpenBuffer1 : BOOL;
	I_PaddleinPosition : BOOL;
	I_BaginIncline : BOOL;
	I_BagatBuffer : BOOL;
	O_RunMotor : BOOL;
	O_OpenBufferStop : BOOL;
	BagSettledBuffer : BOOL;
	BagSettledBufferET : UDINT;
	BagSettled : BOOL;
	BagSettledET : UDINT;
	BagNearTop : BOOL;
	BagNearTopET : UDINT;
	RunOn : BOOL;
	RunOnET : UDINT;
	mySeq : USINT;
	myFirstBag : BOOL;
	O_Select : ARRAY[0..6] OF BOOL;
	ENDI : BOOL;
	O_LineSelect : ARRAY[0..3] OF BOOL;
END_VAR
```

#### 9_spc1Cyclic.ab
```automation-basic
PROGRAM _CYCLIC
	(* cyclic program *)

;----------------------------------------------
;Sequence 10 - SPC1 Pneumatic Conveyor 1 D[910]
;----------------------------------------------

;Inputs
;Incline Conveyor
;-----------------------------------------
;Revision 1.00 09/01/2002 D.J. First Issue
;-----------------------------------------

I_PaddleinPosition		= X[8].X01
I_BaginIncline			= X[8].X02
I_BagatBuffer			= X[3].X01

O_RunMotor 				= FALSE
O_OpenBufferStop		= FALSE
Enable.CDC4Empty       = FALSE

Request.CIC[4]          = FALSE

IF (STEP <5) THEN
	O_LineSelect[2]         = FALSE
	O_LineSelect[1]         = FALSE
ENDIF
//Request.SIC[3]			= FALSE
//Enable.CDC[2]             = FALSE
;Setup Sequence
mySeq                          = 16
;-----------------------
STEP = D[916]
;Setup Pulse contact
PLS = (STEP <> LASTSTEP)
LASTSTEP = STEP

Alarm[mySeq].Name 	= 0
Alarm[mySeq].Bag	= 42
Alarm[mySeq].Beacon	= TRUE
Alarm[mySeq].Extra	= 0
Alarm[mySeq].Time	= 3000
;Run Incline until paddle in position
IF (STEP = 1) THEN
	O_RunMotor = (NOT I_PaddleinPosition)
	IF I_PaddleinPosition THEN
		D[916] = 2
	ENDIF
	Alarm[mySeq].Name = almSwitchFault
ENDIF

;Check romm in buffer
TON_10ms(I_BagatBuffer,300,BagSettledBuffer,BagSettledBufferET)
IF (STEP = 2) THEN
	Request.CIC[4] = (Bag[42].Cat= 0) AND NOT I_BagatBuffer
	IF Request.CDC4Empty AND Request.CIC[4]  AND (D[913] < 5)THEN
		D[916] = 3
	ELSE IF (D[913]	= 5) THEN
		D[916] = 4
	ENDIF
	IF (Request.CIC[4] OR Request.CDC4Empty OR BagSettledBuffer ) THEN
	;	D[916] = 3
	ENDIF
ENDIF

TON_10ms(I_BagatBuffer,300,BagSettledBuffer,BagSettledBufferET)
IF (STEP = 3) THEN
;	Request.CIC[4] = (Bag[42].Cat= 0) AND NOT I_BagatBuffer
		Enable.CDC4Empty  = TRUE
	IF BagSettledBuffer THEN
		D[916] = 4
	ENDIF
ENDIF

TON_10ms(I_BagatBuffer,300,BagSettledBuffer,BagSettledBufferET)
IF (STEP = 4) THEN
;	Enable.CDC4Empty  = TRUE
	IF BagSettledBuffer THEN
			D[916] = 5
	ENDIF
ENDIF

;Wait for bag in incline
IF (STEP = 5) THEN
	;Enable.CDC4Empty  = TRUE
	O_OpenBufferStop = TRUE
	IF I_BaginIncline THEN
		Bag[42].Cat = 0
		D[916] = 6
	ENDIF
	Alarm[mySeq].Name = almSwitchFault

ENDIF

;Let bag settle at base of incline
TON_10ms((STEP = 6),1000,BagSettled,BagSettledET)
IF (STEP = 6) THEN
	IF BagSettled THEN
		D[916] = 7
	ENDIF
ENDIF

IF D[916]<6 THEN
;	O_LineSelect[1] = FALSE
;	O_LineSelect[2] = FALSE
ENDIF

;Move Bag up incline
TON_10ms((STEP = 7),200,BagNearTop,BagNearTopET)
IF (STEP = 7) THEN
	O_RunMotor = TRUE
	IF BagNearTop THEN
		D[916] = 8
	ENDIF
ENDIF

;Wait for Ongoing Sequence to Enable
;Run motor for 0.5 seconds
TON_10ms((STEP = 8),50,RunOn,RunOnET)
IF (STEP = 8) THEN
	O_RunMotor 		= NOT RunOn
	IF Line[11].Clear THEN
		O_LineSelect[1] = TRUE
		C[11]   = 0
		D[916] = 9
	ELSE IF Line[15].Clear THEN
		O_LineSelect[2] = TRUE
		C[15] = 0
		D[916] = 9
	ENDIF
ENDIF

;Run incline until bag at storage lines
IF (STEP = 9) THEN
	O_RunMotor 		= TRUE
		IF (C[11]>0) AND O_LineSelect[1]  THEN
			D[916] = 1
			O_LineSelect[1] = FALSE
		ELSE IF (C[15]>0) AND O_LineSelect[2] THEN
			D[916] = 1
			O_LineSelect[2]
		ENDIF
		Alarm[mySeq].Name = almBagNotArrived
	;Bag in transit arrives at the buffers

ENDIF

;Alarms
TimerAlarm.IN 		= NOT PLS AND (Alarm[mySeq].Name > 0)
TimerAlarm.PT 		= Alarm[mySeq].Time
TimerAlarm FUB TON_10ms()
Alarm[mySeq].On 	= TimerAlarm.Q
Alarm[mySeq].ET 	= TimerAlarm.ET

Y[9].Y14 = O_RunMotor
Y[7].Y12 = O_LineSelect[1]
Y[7].Y13 = O_LineSelect[2]
Y[3].Y03 = O_OpenBufferStop
END_PROGRAM
```

### Program Logical/Sequences/10ms/17_cp12 (IEC) - * SPC1 Empty bags up

#### 9_spc1.var
```iecst
VAR
	I_CarrAtTop : BOOL;
	I_CarrAtBottom : BOOL;
END_VAR
VAR RETAIN
	STEP : UINT;
END_VAR
VAR
	PLS : BOOL;
END_VAR
VAR RETAIN
	LASTSTEP : UINT;
END_VAR
VAR
	O_MoveCarrUp : BOOL;
	O_OpenCarrStop : BOOL;
	O_MoveCarrDown : BOOL;
	I_BagOnCarr : BOOL;
	O_OpenBuffer : BOOL;
	SettledBuffer : BOOL;
	SettledBufferET : TIME;
	I_BagAtBuffer : BOOL;
	BagSettledOnCarr : BOOL;
	BagSettledOnCarrET : TIME;
	I_BagReleased : BOOL;
	TimerAlarm : TON_10ms;
	I_BagAtLLBuff : BOOL;
	O_LLBuffOpen : BOOL;
	SettledBufferSDC2ET : TIME;
	SettledBufferSDC2 : BOOL;
	I_BagAtBufferSDC2 : BOOL;
	Alt : USINT;
	O_OpenBuffer1 : BOOL;
	I_PaddleinPosition : BOOL;
	I_BaginIncline : BOOL;
	I_BagatBuffer : BOOL;
	O_RunMotor : BOOL;
	O_OpenBufferStop : BOOL;
	BagSettledBuffer : BOOL;
	BagSettledBufferET : UDINT;
	BagSettled : BOOL;
	BagSettledET : UDINT;
	BagNearTop : BOOL;
	BagNearTopET : UDINT;
	RunOn : BOOL;
	RunOnET : UDINT;
	mySeq : USINT;
	myFirstBag : BOOL;
	O_Select : ARRAY[0..6] OF BOOL;
	ENDI : BOOL;
	O_LineSelect : ARRAY[0..3] OF BOOL;
	I_BagAtLine1 : BOOL;
	I_BagAtLine2 : BOOL;
	BagAtLine1 : BOOL;
	BagAtLine1ET : UDINT;
	BagAtLine2 : BOOL;
	BagAtLine2ET : UDINT;
	O_SelectLine : ARRAY[0..3] OF BOOL;
END_VAR
```

#### 9_spc1Cyclic.ab
```automation-basic
PROGRAM _CYCLIC
	(* cyclic program *)

;----------------------------------------------
;Sequence 10 - SPC1 Pneumatic Conveyor 1 D[910]
;----------------------------------------------

;Inputs
;Incline Conveyor
;-----------------------------------------
;Revision 1.00 09/01/2002 D.J. First Issue
;-----------------------------------------

I_BagAtLine1		= X[8].X11
I_BagAtLine2		= X[8].X12
//I_BagatBuffer			= X[5].X10

O_RunMotor 				= FALSE
O_OpenBufferStop		= FALSE

O_SelectLine[1]            = FALSE
O_SelectLine[2]            = FALSE
;Setup Sequence
mySeq                          = 17
;-----------------------
STEP = D[917]
;Setup Pulse contact
PLS = (STEP <> LASTSTEP)
LASTSTEP = STEP

;Alarm[mySeq].Name 	= 0
Alarm[mySeq].Bag	= 10016
Alarm[mySeq].Beacon	= TRUE
Alarm[mySeq].Extra	= 0
Alarm[mySeq].Time	= 3000
;wait for space
IF (STEP = 1) THEN
		IF Line[12].Clear THEN
		D[917] = 2
	ENDIF
ENDIF

;Check romm in buffer
TON_10ms(I_BagAtLine1,300,BagAtLine1,BagAtLine1ET)
TON_10ms(I_BagAtLine2,300,BagAtLine2,BagAtLine2ET)
IF (STEP = 2) THEN
	IF Line[12].Clear THEN
		IF BagAtLine1 THEN
			O_SelectLine[1] = TRUE
			C[12]  = 0
			D[917] = 3
		ELSE IF BagAtLine2 THEN
			O_SelectLine[2] = TRUE
			C[12]   = 0
			D[917] = 4
		ENDIF
	ENDIF
ENDIF

;

;Wait for bag in incline
IF (STEP = 3) THEN
	O_SelectLine[1] = TRUE
	IF (C[12]>=1) THEN
		D[917] = 1
	ENDIF
ENDIF

IF (STEP = 4) THEN
	O_SelectLine[2] = TRUE
	IF (C[12]>=1) THEN
		D[917] = 1
	ENDIF
ENDIF

;Alarms
TimerAlarm.IN 		= NOT PLS AND (Alarm[mySeq].Name > 0)
TimerAlarm.PT 		= Alarm[mySeq].Time
TimerAlarm FUB TON_10ms()
Alarm[mySeq].On 	= TimerAlarm.Q
Alarm[mySeq].ET 	= TimerAlarm.ET

Y[8].Y11 = O_SelectLine[1]
Y[8].Y12 = O_SelectLine[2]
END_PROGRAM
```

### Program Logical/Sequences/10ms/18_cdc8 (IEC) - * SDC1 Machine 1 BCD/CAN

#### 6_sdc1.var
```iecst
VAR RETAIN
	STEP : UINT;
	PLS : BOOL;
	LASTSTEP : UINT;
	SteadyUp : BOOL;
	CloserUpET : TIME;
	SteadysDown : BOOL;
	SteadysDownET : TIME;
	LoadDropped : BOOL;
END_VAR
VAR
	SteadyUpET : TIME;
	CloserDownET : TIME;
	SettledAtDischargerET : TIME;
	MinOpenET : TIME;
	SettledAtDischarger : BOOL;
	CloserDown : BOOL;
	MinOpen : BOOL;
	CloserUp : BOOL;
	SettledAtBuffer : BOOL;
	SettledAtBufferET : TIME;
	I_BagAtBuffer : BOOL;
	O_OpenStop : BOOL;
	O_OpenBag : BOOL;
	O_Steadys : BOOL;
	O_OpenBuffer : BOOL;
	O_Closer : BOOL;
	I_BagAtDischarger : BOOL;
	I_OpenBag : BOOL;
	I_LoadDropped : BOOL;
	TestDrop : BOOL;
	DischargerEnable : BOOL;
	TestDischarger : BOOL;
	Remainder : SINT;
	TimerAlarm : TON_10ms;
	WgtRound : UINT;
	a : BOOL;
	I_BagEmpty : BOOL;
	MySeq : USINT;
	O_BagReady : BOOL;
	I_BagOut : BOOL;
END_VAR
```

#### 6_sdc1Cyclic.ab
```automation-basic
PROGRAM _CYCLIC
	(* cyclic program *)

;Sequence 6 - Discharger 1 D[906]
a

;-----------------------------------------
;Revision 1.00 19/12/2005 D.J. First Issue
;-----------------------------------------

DischargerEnable 		= ((D[18] > 0) AND NOT Std.HaltSys)
MySeq                       = 18

I_BagAtBuffer			  = X[4].X03
I_BagAtDischarger = X[3].X02
//I_SafetyRunning       = X[8].X15

I_OpenBag				= X[3].X16 OR TestDrop           ;X[23].X01
//I_LoadDropped			= X[7].X13 OR TestDischarger  ;X[23].X02
I_BagOut              = X[8].X10
I_BagEmpty          = X[2].X09

O_Steadys				= FALSE ;Y[6].Y01
O_OpenBuffer 			= FALSE ;Y[6].Y02
O_OpenBag				= FALSE ;Y[6].Y03
O_OpenStop				= FALSE ;Y[6].Y04
O_Closer				= FALSE ;Y[6].Y05
O_BagReady          = FALSE

;Alarm
Alarm[MySeq].Name 			= 0 ;Clear sequence alarm name
Alarm[MySeq].Bag 			= 46
Alarm[MySeq].Beacon			= TRUE
Alarm[MySeq].Extra			= 0
Alarm[MySeq].Time			= 3000

;Setup Sequence
STEP = D[900+MySeq]
;Setup Pulse contact
PLS = (STEP <> LASTSTEP)
LASTSTEP = STEP

;Step 0 - Disabled
IF (STEP = 0) THEN
	;Disabled
ENDIF

;Check Status - Bag settled at buffer, no bag at discharger, bag at buffer on screen and no bag at discharger on the screen
TON_10ms(I_BagAtBuffer,300,SettledAtBuffer,SettledAtBufferET)
IF (STEP = 1) THEN
	IF DischargerEnable AND SettledAtBuffer AND  NOT I_BagAtDischarger AND (Bag[49].Cat = 0) AND (Bag[78].Cat > 0)THEN
		D[900+MySeq] = 2
	ENDIF
	IF (Bag[49].Cat > 0) THEN
		Alarm[MySeq].Name = almBagDataError
	ELSE IF I_BagAtDischarger THEN
		Alarm[MySeq].Name = almSwitchFault
	ENDIF
ENDIF

;Wait for bag in discharger
IF (STEP = 2) THEN
	O_OpenBuffer 	= TRUE

	IF I_BagAtDischarger THEN
		D[900+MySeq] = 3
	ENDIF
	Alarm[7].Name = almBagNotArrived
ENDIF

;Let bag settle in discharger
TON_10ms(((STEP = 3) AND I_BagAtDischarger),1000,SettledAtDischarger,SettledAtDischargerET)
IF (STEP = 3) THEN
	IF (Bag[49].Cat = 0) AND (Bag[78].Cat>0) THEN
		Bag[49] = Bag[78]
		Bag[78]   = Bag[0]
	ENDIF
	IF SettledAtDischarger THEN
		D[900+MySeq] = 4
	ENDIF
	Alarm[MySeq].Name = almBagNotSettled
ENDIF

;Allow steadys to move down
TON_10ms((STEP = 4),400,SteadysDown,SteadysDownET)
IF (STEP = 4) THEN
	IF SteadysDown AND (Bag[49].Cat <> Std.MaxCats)  THEN
		D[900+MySeq] = 5
	ENDIF
	IF (Bag[49].Cat = Std.MaxCats) AND SteadysDown THEN
		D[900+MySeq] = 8
	ENDIF
ENDIF

;Steady cylinders on from steps 4 - 9
O_Steadys = ((STEP >= 4) AND (STEP <= 9))

;Bag opener on from step 5 - 8
O_OpenBag = ((STEP >= 6) AND (STEP <= 8))

;Wash Codes
;IF (STEP = 4) OR (STEP = 5) THEN
;
;;round up weight to give to wash machine
;	Remainder = SINT(Bag[228].Wgt MOD 10)
;	IF (Remainder > 4) THEN
;		WgtRound = (Bag[228].Wgt + 10)
;	ELSE
;		WgtRound = Bag[228].Wgt
;	ENDIF
;
;
;;Codes to CBW
;	CAN[1].Category = Bag[228].Cat
;	CAN[1].Customer = Bag[228].Cus
;	CAN[1].Weight   = (WgtRound / 10)
;ELSE
;	CAN[1].Category = 0
;	CAN[1].Customer = 0
;	CAN[1].Weight   = 0
;ENDIF

;Bag Ready to Washing Machine
IF (STEP = 5) THEN
	O_BagReady = TRUE
	O_Closer        = TRUE
	IF I_OpenBag OR TestDischarger THEN
		D[900+MySeq] = 6
	ENDIF

ENDIF

;Open Bag Until LoadDropped recieved and has been open for 6 seconds
TON_10ms((STEP = 6) AND NOT I_BagEmpty,300,MinOpen,MinOpenET) ;ET means Elapsed Time
IF (STEP = 6) THEN
	IF I_OpenBag THEN
		LoadDropped = TRUE
	ENDIF
	IF (NOT I_OpenBag AND MinOpen) THEN
		D[900+MySeq] = 7
	ENDIF
	Alarm[MySeq].Name = almLoadNotDropped
	ELSE
	LoadDropped = FALSE
ENDIF

;Change display to empty bag
IF (STEP = 7) THEN
	O_BagReady = TRUE
	IF I_OpenBag THEN
		LoadDropped = TRUE
	ENDIF
	IF (LoadDropped  OR TestDrop) THEN ;AND I_BagEmpty) OR TestDrop) THEN
		Bag[49].Cat 	= Std.MaxCats
		D[900+MySeq] 			= 8
	ENDIF
	Alarm[MySeq].Name = almGeneralSequence
	ELSE
	LoadDropped = FALSE
ENDIF

;Close bag
TON_10ms((STEP = 8),700,CloserDown,CloserDownET)
IF (STEP = 8) THEN
	O_Closer = TRUE
	IF CloserDown THEN
		D[900+MySeq] = 9
	ENDIF
ENDIF

;Allow closer to go back up
TON_10ms((STEP = 9),700,CloserUp,CloserUpET)
IF (STEP = 9) THEN
	IF CloserUp THEN
		D[900+MySeq] = 10
	ENDIF
ENDIF

;Allow steadys to go up
TON_10ms((STEP = 10),400,SteadyUp,SteadyUpET)
IF (STEP = 10) THEN
	IF SteadyUp THEN
		D[900+MySeq] = 11
	ENDIF
ENDIF

;Check for space on empty bag buffer
IF (STEP = 11) THEN

	IF (D[922]=3) AND NOT X[8].X07  THEN
		D[900+MySeq] = 12
	ENDIF

ENDIF

;Open buffer stop - unitl bag out
IF (STEP = 12) THEN
	O_OpenStop = TRUE
	IF PLS THEN
		;C[14] = 0
	ENDIF
	Bag[49].Cat = 0
	Bag[49].Cus = 0
	Bag[49].Wgt = 0
	IF I_BagOut  THEN
		D[900+MySeq] = 1
	ENDIF
	Alarm[MySeq].Name = almBagNotReleased
ENDIF

;Alarms
TimerAlarm.IN 	= NOT PLS AND (Alarm[MySeq].Name > 0)
TimerAlarm.PT 	= Alarm[MySeq].Time
TimerAlarm FUB TON_10ms()
Alarm[MySeq].On 	= TimerAlarm.Q
Alarm[MySeq].ET 	= TimerAlarm.ET

;Outputs

Y[6].Y01 = O_BagReady
Y[4].Y05 = O_OpenBuffer
Y[5].Y06 = O_Steadys
Y[5].Y08 = O_OpenBag
Y[5].Y07 = O_OpenStop
Y[5].Y09 = O_Closer

END_PROGRAM
```

### Program Logical/Sequences/10ms/19_cp13 (IEC) - * SPC1 Empty bags up

#### 9_spc1.var
```iecst
VAR
	I_CarrAtTop : BOOL;
	I_CarrAtBottom : BOOL;
END_VAR
VAR RETAIN
	STEP : UINT;
END_VAR
VAR
	PLS : BOOL;
END_VAR
VAR RETAIN
	LASTSTEP : UINT;
END_VAR
VAR
	O_MoveCarrUp : BOOL;
	O_OpenCarrStop : BOOL;
	O_MoveCarrDown : BOOL;
	I_BagOnCarr : BOOL;
	O_OpenBuffer : BOOL;
	SettledBuffer : BOOL;
	SettledBufferET : TIME;
	I_BagAtBuffer : BOOL;
	BagSettledOnCarr : BOOL;
	BagSettledOnCarrET : TIME;
	I_BagReleased : BOOL;
	TimerAlarm : TON_10ms;
	I_BagAtLLBuff : BOOL;
	O_LLBuffOpen : BOOL;
	SettledBufferSDC2ET : TIME;
	SettledBufferSDC2 : BOOL;
	I_BagAtBufferSDC2 : BOOL;
	Alt : USINT;
	O_OpenBuffer1 : BOOL;
	I_PaddleinPosition : BOOL;
	I_BaginIncline : BOOL;
	I_BagatBuffer : BOOL;
	O_RunMotor : BOOL;
	O_OpenBufferStop : BOOL;
	BagSettledBuffer : BOOL;
	BagSettledBufferET : UDINT;
	BagSettled : BOOL;
	BagSettledET : UDINT;
	BagNearTop : BOOL;
	BagNearTopET : UDINT;
	RunOn : BOOL;
	RunOnET : UDINT;
	mySeq : USINT;
	myFirstBag : BOOL;
	O_Select : ARRAY[0..6] OF BOOL;
	ENDI : BOOL;
	O_LineSelect : ARRAY[0..3] OF BOOL;
	I_BagAtLine1 : BOOL;
	I_BagAtLine2 : BOOL;
	BagAtLine1 : BOOL;
	BagAtLine1ET : UDINT;
	BagAtLine2 : BOOL;
	BagAtLine2ET : UDINT;
	O_SelectLine : ARRAY[0..3] OF BOOL;
	I_BagInCPC1 : BOOL;
	O_Reset : BOOL;
	Reset : BOOL;
	ResetET : UDINT;
	BagSettledAtBuffer : BOOL;
	BagSettledAtBufferET : UDINT;
	Destination : BOOL;
	O_SelectY706 : BOOL;
	O_SelectY510 : BOOL;
	O_SelectY514 : BOOL;
END_VAR
```

#### 9_spc1Cyclic.ab
```automation-basic
PROGRAM _CYCLIC
	(* cyclic program *)

;----------------------------------------------
;Sequence 10 - SPC1 Pneumatic Conveyor 1 D[910]
;----------------------------------------------

;Inputs
;Incline Conveyor
;-----------------------------------------
;Revision 1.00 09/01/2002 D.J. First Issue
;-----------------------------------------

I_BagAtBuffer		= X[5].X02
I_BagInCPC1  		= X[2].X04
//I_BagatBuffer			= X[5].X10

O_RunMotor 				= FALSE
O_OpenBufferStop		= FALSE
O_Reset                     = FALSE

O_SelectY510 			= FALSE
O_SelectY514            = FALSE
O_SelectY706            = FALSE
mySeq                          = 19
;-----------------------
STEP = D[919]
;Setup Pulse contact
PLS = (STEP <> LASTSTEP)
LASTSTEP = STEP

;Alarm[mySeq].Name 	= 0
Alarm[mySeq].Bag	= 51
Alarm[mySeq].Beacon	= TRUE
Alarm[mySeq].Extra	= 0
Alarm[mySeq].Time	= 3000
;wait for space
TON_10ms((STEP = 1),300,Reset,ResetET)
IF (STEP = 1) THEN
		O_Reset  = TRUE
		IF Reset THEN
		D[919] = 2
	ENDIF
ENDIF

;Check romm in buffer
TON_10ms(I_BagAtBuffer,300,BagSettledAtBuffer,BagSettledAtBufferET)

IF (STEP = 2) THEN
	IF (Bag[51].Cat>0) THEN
		IF (Line[Bag[51].Dst].Space>0) AND (Bag[60].Cat=0) THEN
			D[919] = 3
		ENDIF
	ENDIF
ENDIF

;

;Wait for bag in incline
IF (STEP = 3) THEN
	IF BagSettledAtBuffer THEN
		IF (Bag[51].Dst >= 1) AND (Bag[51].Dst <=4) THEN
			IF (Bag[36].Cat=0) AND Request.CP[5]  THEN
				D[919]=4
			ENDIF
		ELSE IF Line[8].Clear AND (D[920]=3)	AND X[2].X01 AND (Bag[51].Dst = 8) THEN
			D[919] = 5
		ELSE IF (Bag[51].Dst = 5) AND Line[5].Clear AND (Bag[29].Cat=0)  THEN
			C[5] = 0
			D[919] = 6
		ELSE IF (Bag[51].Dst = 6) AND Line[6].Clear AND (Bag[24].Cat=0)  THEN
			C[6] = 0
			D[919]= 7
		ENDIF
	ENDIF
ENDIF

;move to CIC1
IF (STEP = 4) THEN
		O_OpenBufferStop = TRUE

		IF NOT Request.CP[5]  THEN
			IF (Bag[51].Cat>0) AND (Bag[36].Cat=0) THEN
				Bag[36] = Bag[51]
				Bag[51] = Bag[0]
			ENDIF
			D[919] = 1
		ENDIF
ENDIF

IF (STEP = 5) THEN
	IF PLS THEN
		IF (Bag[51].Cat>0) AND (Bag[60].Cat=0) THEN
				Bag[60] = Bag[51]
				Bag[51] = Bag[0]
			ENDIF
		ENDIF
		O_OpenBufferStop = TRUE
		O_SelectY706        = TRUE
		O_SelectY510        = TRUE
		IF I_BagInCPC1 THEN
			IF (Bag[60].Cat>0) AND (Bag[58].Cat=0) THEN
				Bag[58] = Bag[60]
				Bag[60] = Bag[0]
			ENDIF
			D[919] = 1
		ENDIF
ENDIF

IF (STEP = 6) THEN
	IF PLS THEN
		IF (Bag[51].Cat>0) AND (Bag[60].Cat=0) THEN
				Bag[60] = Bag[51]
				Bag[51] = Bag[0]
			ENDIF
		ENDIF
		O_OpenBufferStop = TRUE
		O_SelectY514        = TRUE
		O_SelectY510        = TRUE
	IF Line[5].Trip THEN
		IF (Bag[60].Cat>0) AND (Bag[29].Cat=0) THEN
				Bag[29] = Bag[60]
				Bag[60] = Bag[0]
			ENDIF
			D[919] = 1
		ENDIF
//	ENDIF
ENDIF

IF (STEP = 7) THEN
	IF PLS THEN
		IF (Bag[51].Cat>0) AND (Bag[60].Cat=0) THEN
				Bag[60] = Bag[51]
				Bag[51] = Bag[0]
		ENDIF
	 ENDIF
		O_OpenBufferStop = TRUE
	//	O_SelectY514        = TRUE
		O_SelectY510        = TRUE
	IF Line[6].Trip THEN
		IF (Bag[60].Cat>0) AND (Bag[24].Cat=0) THEN
				Bag[24] = Bag[60]
				Bag[60] = Bag[0]
				Bag[24].Dst = 0
		ENDIF
			D[919] = 1
	ENDIF
//	ENDIF
ENDIF

;Alarms
TimerAlarm.IN 		= NOT PLS AND (Alarm[mySeq].Name > 0)
TimerAlarm.PT 		= Alarm[mySeq].Time
TimerAlarm FUB TON_10ms()
Alarm[mySeq].On 	= TimerAlarm.Q
Alarm[mySeq].ET 	= TimerAlarm.ET

Y[5].Y11  =  O_Reset
Y[5].Y15  =  O_Reset
Y[7].Y08  =  O_Reset

Y[9].Y12 = O_OpenBufferStop
Y[5].Y10 = O_SelectY510
Y[5].Y14 = O_SelectY514
Y[7].Y06 = O_SelectY706
END_PROGRAM
```

### Program Logical/Sequences/10ms/20_cpc1 (IEC, version 1.00.0) - * SPC1 Empty bags up

#### 9_spc1Cyclic.ab
```automation-basic
PROGRAM _CYCLIC
	(* cyclic program *)

;----------------------------------------------
;Sequence 10 - SPC1 Pneumatic Conveyor 1 D[910]
;----------------------------------------------

;Inputs
;Incline Conveyor
;-----------------------------------------
;Revision 1.00 09/01/2002 D.J. First Issue
;-----------------------------------------

I_CarrAtTop				= X[2].X01
I_CarrAtBottom			= X[2].X02
I_BagOnCarr				= X[2].X03
I_BagArrived            = X[2].X04
I_BagInCIC6             = X[6].X14

O_MoveCarrUp			= FALSE
O_MoveCarrDown			= FALSE
O_OpenCarrStop			= FALSE
O_RailEndStop           = FALSE

mySeq                          = 5
;-----------------------
STEP = D[920]
;Setup Pulse contact
PLS = (STEP <> LASTSTEP)
LASTSTEP = STEP

;Alarm[mySeq].Name 	= 0
Alarm[mySeq].Bag	= 58
Alarm[mySeq].Beacon	= TRUE
Alarm[mySeq].Extra	= 0
Alarm[mySeq].Time	= 3000
;Run Incline until paddle in position
IF (STEP = 1) THEN
	O_MoveCarrUp = TRUE
	IF I_CarrAtTop THEN
		D[920] = 2
	ENDIF
ENDIF

;Check romm in buffer
TON_10ms(I_BagatBuffer,300,BagSettledBuffer,BagSettledBufferET)
;Check Status
IF (STEP = 2) THEN
	O_MoveCarrUp = TRUE
	IF (NOT I_BagOnCarr AND (Bag[58].Cat = 0)) THEN
		D[920] = 3
	ENDIF
ENDIF

;

;Wait for bag in incline

IF (STEP = 3) THEN
	O_MoveCarrUp = TRUE
    O_RailEndStop = TRUE
   IF I_BagOnCarr THEN
	D[920] = 4
   ENDIF
ENDIF

;Let bag settle on carriage
TON_10ms(I_BagOnCarr,500,BagSettledOnCarr,BagSettledOnCarrET)
IF (STEP = 4) THEN
    O_RailEndStop = TRUE
	O_MoveCarrUp = TRUE
	IF (BagSettledOnCarr) THEN
		D[920] = 5
	ENDIF
ENDIF

;Check top switch
IF (STEP = 5) THEN
	O_MoveCarrUp = TRUE
	IF NOT I_CarrAtBottom THEN
		D[920] = 6
	ENDIF
ENDIF

;Move Carriage up to top position
IF (STEP = 6) THEN
	O_MoveCarrDown = TRUE
	IF I_CarrAtBottom THEN
		D[920] = 7
	ENDIF
ENDIF

;Check Destination Of Bag
IF (STEP = 7) THEN
	   O_MoveCarrDown 	= TRUE
		IF ((D[921] = 3) AND (Bag[59].Cat = 0)) THEN
		D[920]  = 8
	ENDIF
ENDIF

;Set LoadDropped to False
IF (STEP <> 8) THEN
	BagInCIC6 = FALSE
ENDIF

;Run incline conveyor until bag at destination
IF (STEP = 8) THEN
	O_OpenCarrStop 	= TRUE
    O_MoveCarrDown 	= TRUE
	IF I_BagInCIC6 THEN
		BagInCIC6 = TRUE
	ENDIF
	IF (BagInCIC6) THEN
		IF (Bag[58].Cat>0) AND (Bag[59].Cat=0) THEN
				Bag[59] = Bag[58]
				Bag[58] = Bag[0]
			ENDIF
		D[920] = 9
	ENDIF
ENDIF

;Check Bottom position switch
IF (STEP = 9) THEN
	O_MoveCarrDown 	= TRUE
	IF NOT I_CarrAtTop AND NOT I_BagOnCarr THEN
		D[920] = 1
	ENDIF
ENDIF

;Alarms
TimerAlarm.IN 		= NOT PLS AND (Alarm[mySeq].Name > 0)
TimerAlarm.PT 		= Alarm[mySeq].Time
TimerAlarm FUB TON_10ms()
Alarm[mySeq].On 	= TimerAlarm.Q
Alarm[mySeq].ET 	= TimerAlarm.ET

;Outputs
Y[2].Y01 = O_MoveCarrUp
Y[2].Y02 = O_MoveCarrDown
Y[2].Y04 = O_RailEndStop
Y[2].Y03 = (O_OpenCarrStop 	AND O_MoveCarrDown)

END_PROGRAM
```

#### 9_spc1.var
```iecst
VAR
	I_CarrAtTop : BOOL;
	I_CarrAtBottom : BOOL;
END_VAR
VAR RETAIN
	STEP : UINT;
END_VAR
VAR
	PLS : BOOL;
END_VAR
VAR RETAIN
	LASTSTEP : UINT;
END_VAR
VAR
	O_MoveCarrUp : BOOL;
	O_OpenCarrStop : BOOL;
	O_MoveCarrDown : BOOL;
	I_BagOnCarr : BOOL;
	O_OpenBuffer : BOOL;
	SettledBuffer : BOOL;
	SettledBufferET : TIME;
	I_BagAtBuffer : BOOL;
	BagSettledOnCarr : BOOL;
	BagSettledOnCarrET : TIME;
	I_BagReleased : BOOL;
	TimerAlarm : TON_10ms;
	I_BagAtLLBuff : BOOL;
	O_LLBuffOpen : BOOL;
	SettledBufferSDC2ET : TIME;
	SettledBufferSDC2 : BOOL;
	I_BagAtBufferSDC2 : BOOL;
	Alt : USINT;
	O_OpenBuffer1 : BOOL;
	I_PaddleinPosition : BOOL;
	I_BaginIncline : BOOL;
	I_BagatBuffer : BOOL;
	O_RunMotor : BOOL;
	O_OpenBufferStop : BOOL;
	BagSettledBuffer : BOOL;
	BagSettledBufferET : UDINT;
	BagSettled : BOOL;
	BagSettledET : UDINT;
	BagNearTop : BOOL;
	BagNearTopET : UDINT;
	RunOn : BOOL;
	RunOnET : UDINT;
	mySeq : USINT;
	myFirstBag : BOOL;
	O_Select : ARRAY[0..6] OF BOOL;
	ENDI : BOOL;
	I_BagArrived : BOOL;
	I_BagInCIC6 : BOOL;
	O_RailEndStop : BOOL;
	BagInCIC6 : BOOL;
END_VAR
```

### Program Logical/Sequences/10ms/21_cic6 (IEC) - * SPC1 Empty bags up

#### 9_spc1Cyclic.ab
```automation-basic
PROGRAM _CYCLIC
	(* cyclic program *)

;----------------------------------------------
;Sequence 10 - SPC1 Pneumatic Conveyor 1 D[910]
;----------------------------------------------

;Inputs
;Incline Conveyor
;-----------------------------------------
;Revision 1.00 09/01/2002 D.J. First Issue
;-----------------------------------------

I_PaddleinPosition		= X[6].X09
I_BaginIncline			= X[6].X14

O_RunMotor 				= FALSE

O_OpenBufferStop		= FALSE

Request.CIC[1]			= FALSE

;Setup Sequence
;-----------------------
STEP = D[921]
;Setup Pulse contact
PLS = (STEP <> LASTSTEP)
LASTSTEP = STEP

;Alarm
;TON_10ms(((NOT PLS) AND (STEP = 3)),1000,Alarm[9],AlarmET[9])

;Run Incline until paddle in position
IF (STEP = 1) THEN
	O_RunMotor = (NOT I_PaddleinPosition)
	IF I_PaddleinPosition THEN
		D[921] = 2
	ENDIF
ENDIF

;Check romm in buffer
TON_10ms(I_BagatBuffer,300,BagSettledBuffer,BagSettledBufferET)
IF (STEP = 2) THEN
	IF NOT ((I_BaginIncline) AND (Bag[59].Cat = 0)) THEN
		D[921] = 3

	ENDIF
ENDIF

;

;Wait for bag in incline
IF (STEP = 3) THEN
IF I_BaginIncline AND (Bag[59].Cat > 0) THEN
		D[921] = 4
	ENDIF
ENDIF

;Let bag settle at base of incline
TON_10ms((STEP = 4),1000,BagSettled,BagSettledET)
IF (STEP = 4) THEN
	IF BagSettled THEN
		D[921] = 5
	ENDIF
ENDIF

;Move Bag up incline
TON_10ms((STEP = 5),200,BagNearTop,BagNearTopET)
IF (STEP = 5) THEN
	O_RunMotor = TRUE
	IF BagNearTop THEN
		D[921] = 6
	ENDIF
ENDIF

;Wait for Ongoing Sequence to Enable
;Run motor for 0.5 seconds
TON_10ms((STEP = 6),50,RunOn,RunOnET)
IF (STEP = 6) THEN
	O_RunMotor 		= NOT RunOn
	IF ((Line[8].Clear) AND (Bag[81].Cat = 0)) THEN
		C[8] = 0
		D[921]  = 7
	ENDIF
ENDIF

;Run incline until bag at storage lines
IF (STEP = 7) THEN
	O_RunMotor 		= TRUE
	IF Line[8].Full THEN
        IF (Bag[59].Cat>0)AND (Bag[81].Cat=0)THEN
				Bag[81] = Bag[59]
				Bag[59] = Bag[0]
		ENDIF
		D[921] = 1
	ENDIF
ENDIF

Y[8].Y10 = O_RunMotor

END_PROGRAM
```

### Program Logical/Sequences/10ms/22_cic7 (IEC, version 1.00.0) - * SPC1 Empty bags up

#### 9_spc1Cyclic.ab
```automation-basic
PROGRAM _CYCLIC
	(* cyclic program *)

;----------------------------------------------
;Sequence 10 - SPC1 Pneumatic Conveyor 1 D[910]
;----------------------------------------------

;Inputs
;Incline Conveyor
;-----------------------------------------
;Revision 1.00 09/01/2002 D.J. First Issue
;-----------------------------------------

I_PaddleinPosition		= X[8].X03
I_BaginIncline			= X[8].X07
I_BagOut                = X[4].X08

Request.CIC[7]            = FALSE

O_RunMotor 				= FALSE

;Setup Sequence
;-----------------------
STEP = D[922]
;Setup Pulse contact
PLS = (STEP <> LASTSTEP)
LASTSTEP = STEP

;Alarm
;TON_10ms(((NOT PLS) AND (STEP = 3)),1000,Alarm[9],AlarmET[9])

;Run Incline until paddle in position
IF (STEP = 1) THEN
	O_RunMotor = (NOT I_PaddleinPosition)
	IF I_PaddleinPosition THEN
		D[922] = 2
	ENDIF
ENDIF

;Check romm in buffer
TON_10ms(I_BagatBuffer,300,BagSettledBuffer,BagSettledBufferET)
IF (STEP = 2) THEN
	//IF NOT ((I_BaginIncline) AND (Bag[59].Cat = 0)) THEN
		D[922] = 3

	//ENDIF
ENDIF

;

;Wait for bag in incline
IF (STEP = 3) THEN
IF I_BaginIncline  THEN
		D[922] = 4
	ENDIF
ENDIF

;Let bag settle at base of incline
TON_10ms((STEP = 4),1000,BagSettled,BagSettledET)
IF (STEP = 4) THEN
	IF BagSettled THEN
		D[922] = 5
	ENDIF
ENDIF

;Move Bag up incline
TON_10ms((STEP = 5),200,BagNearTop,BagNearTopET)
IF (STEP = 5) THEN
	O_RunMotor = TRUE
	IF BagNearTop THEN
		D[922] = 6
	ENDIF
ENDIF

;Wait for Ongoing Sequence to Enable
;Run motor for 0.5 seconds
TON_10ms((STEP = 6),50,RunOn,RunOnET)
IF (STEP = 6) THEN
	O_RunMotor 	= NOT RanOn
    Request.CIC[7] = TRUE
	IF Enable.CIC[7] THEN
		D[922] = 7

	ENDIF
ENDIF

;Run incline until bag at storage lines
IF (STEP = 7) THEN
	O_RunMotor 		= TRUE
	IF I_BagOut THEN
		D[922] = 1
	ENDIF

ENDIF

Y[8].Y13 = O_RunMotor

END_PROGRAM
```

#### 9_spc1.var
```iecst
VAR
	I_CarrAtTop : BOOL;
	I_CarrAtBottom : BOOL;
END_VAR
VAR RETAIN
	STEP : UINT;
END_VAR
VAR
	PLS : BOOL;
END_VAR
VAR RETAIN
	LASTSTEP : UINT;
END_VAR
VAR
	O_MoveCarrUp : BOOL;
	O_OpenCarrStop : BOOL;
	O_MoveCarrDown : BOOL;
	I_BagOnCarr : BOOL;
	O_OpenBuffer : BOOL;
	SettledBuffer : BOOL;
	SettledBufferET : TIME;
	I_BagAtBuffer : BOOL;
	BagSettledOnCarr : BOOL;
	BagSettledOnCarrET : TIME;
	I_BagReleased : BOOL;
	TimerAlarm : TON_10ms;
	I_BagAtLLBuff : BOOL;
	O_LLBuffOpen : BOOL;
	SettledBufferSDC2ET : TIME;
	SettledBufferSDC2 : BOOL;
	I_BagAtBufferSDC2 : BOOL;
	Alt : USINT;
	O_OpenBuffer1 : BOOL;
	I_PaddleinPosition : BOOL;
	I_BaginIncline : BOOL;
	I_BagatBuffer : BOOL;
	O_RunMotor : BOOL;
	O_OpenBufferStop : BOOL;
	BagSettledBuffer : BOOL;
	BagSettledBufferET : UDINT;
	BagSettled : BOOL;
	BagSettledET : UDINT;
	BagNearTop : BOOL;
	BagNearTopET : UDINT;
	RunOn : BOOL;
	RunOnET : UDINT;
	O_Select : ARRAY[0..6] OF BOOL;
	I_BagOut : BOOL;
	RanOn : BOOL;
END_VAR
```

### Program Logical/Sequences/10ms/23_Ebag (IEC) - *PP4 Full bag from PID4

#### pp.var
```iecst
VAR
	BagReleased : BOOL;
	BagValid : BOOL;
	DestValid : BOOL;
	I_BagAtSep : BOOL;
	I_BagInSep : BOOL;
END_VAR
VAR RETAIN
	LASTSTEP : UINT;
END_VAR
VAR
	LineValid : ARRAY[0..2] OF BOOL;
	myBag : UINT;
	myDest : USINT;
	myIO : UINT;
	myIO2 : UINT;
	myPrevSelLine : USINT;
	myRelLastBag : ARRAY[0..2] OF UINT;
	myRelLine : ARRAY[0..2] OF UINT;
	mySelLine : USINT;
	mySeq : UINT;
	myZone : INT;
	O_OpenSep : BOOL;
	O_Select : ARRAY[0..2] OF BOOL;
END_VAR
VAR RETAIN
	PLS : BOOL;
END_VAR
VAR
	PointsReset : BOOL;
	PointsResetET : UDINT;
	ResetPoints : BOOL;
	SettledAtSep : BOOL;
	SettledAtSepET : UDINT;
END_VAR
VAR RETAIN
	STEP : UINT;
END_VAR
VAR
	TimerAlarm : TON_10ms;
	SettledInSep : BOOL;
	SettledInSepET : UDINT;
	BagInSep : BOOL;
	Reset : BOOL;
	ResetET : UDINT;
	O_Reset : BOOL;
END_VAR
```

#### pp.ab
```automation-basic
;--------------------------------------------
;Sequence 0 - XXX0  D[900 + mySeq]
;--------------------------------------------

PROGRAM _INIT
(* init program *)
END_PROGRAM

PROGRAM _CYCLIC

;Inputs
mySeq				= 23	;Sequence number

Enable.CIC[1]       = FALSE

myZone	= 0

Enable.CIC[8]		= FALSE

Alarm[mySeq].Name 	= 0
Alarm[mySeq].Bag	= 0
Alarm[mySeq].Beacon	= TRUE
Alarm[mySeq].Extra	= 0
Alarm[mySeq].Time	= 3000

;Setup Sequence
STEP = D[900 + mySeq]
;Setup Pulse contact
PLS = (STEP <> LASTSTEP)
LASTSTEP = STEP

;Sequence
IF (STEP = 0) THEN
	;Disabled
ENDIF
;Reset Points
TON_10ms((STEP = 1),250,Reset,ResetET)
IF (STEP = 1) THEN
	O_Reset = NOT Reset
    D[52] = 0
	IF Reset AND Line[14].Clear THEN
		D[923] = 2
	ENDIF
;	Alarm[mySeq].Name 	= almSwitchFault
ENDIF

;Decide where to take bag from
IF (STEP = 2) THEN
	IF (D[915] = 11) THEN   ;Empty bag from CDC7
		D[52]	= 3
		C[14]	= 0
		D[923]	= 3
	ELSE IF (Request.CIC[8]) THEN   ;Empty bag from CIC8
		D[52]	= 4
		C[14]	= 0
		D[923]	= 4
	ENDIF
ENDIF

;Enable CDC7 to release bag
IF (STEP = 3) THEN
    ;Enable.CP5      = (D[49] = 3)
    IF (D[915] = 11) THEN
    	D[915] = 12
    ENDIF
	IF Line[14].Full THEN
		D[923] = 1
	ENDIF
ENDIF

;Enable CIC8 to release bag
IF (STEP = 4) THEN
    Enable.CIC[8] = (D[52] = 4)
	IF Line[14].Full THEN
		D[923] = 1
	ENDIF
ENDIF

Y[2].Y09 = O_Reset

;Alarms
TimerAlarm.IN 		= NOT PLS AND (Alarm[mySeq].Name > 0)
TimerAlarm.PT 		= Alarm[mySeq].Time
TimerAlarm FUB TON_10ms()
Alarm[mySeq].On 	= TimerAlarm.Q
Alarm[mySeq].ET 	= TimerAlarm.ET
//Alarm[mySeq].Zone 	= myZone
END_PROGRAM
```

### Program Logical/Sequences/10ms/24_csb1 (IEC, version 1.00.0) - * SVC1 Inverter VC

#### 7_svc1Cyclic.ab
```automation-basic
PROGRAM _CYCLIC
	(* cyclic program *)
DDDDDD

I_OpenBag				= X[4].X07

I_DischBagOpened		= (D[915] = 6)

O_BagReady				= FALSE
O_OpenCatch				= FALSE
O_OpenBag				= FALSE
O_CloseBag				= FALSE

Enable.CDC[7]		    = FALSE

mySeq				= 24	;Sequence number

Alarm[mySeq].Name 	= 0
Alarm[mySeq].Bag	= 0
Alarm[mySeq].Beacon	= TRUE
Alarm[mySeq].Extra	= 0
Alarm[mySeq].Time	= 3000
;Setup Sequence
;-----------------------
STEP = D[924]
;Setup Pulse contact
PLS = (STEP <> LASTSTEP)
LASTSTEP = STEP

;Alarm
;TON_10ms(((NOT PLS) AND (STEP = 6)),6000,Alarm[8],AlarmET[8])

;Step 0 - Disabled
IF (STEP = 0) THEN
	;Disabled
ENDIF

;Wait for bag on carriage
IF (STEP = 1) THEN
	IF (NOT I_OpenBag) THEN
		D[924] = 2
	ENDIF
ENDIF

;Step 2 - Enable discharger to open
TON_10ms(I_DischBagOpened,600,TopBagOpen,TopBagOpenET)
IF (STEP = 2) THEN
	Enable.CDC[7] = I_OpenBag
	O_BagReady = (D[915] = 5)
	IF I_OpenBag THEN
		OpenCatch = TRUE
	ENDIF
	O_OpenCatch = OpenCatch
	IF TopBagOpen THEN
		D[924] 		= 3
	ENDIF
	ELSE
	OpenCatch = FALSE
ENDIF

;Step 3 - Bag being loaded
IF (STEP = 3) THEN
		O_BagReady = Std.Clock500ms
		O_OpenCatch = TRUE
		IF I_OpenBag THEN
			BagClear = TRUE
		ENDIF
		IF BagClear AND NOT I_OpenBag THEN
			D[924] = 4
		ENDIF
	ELSE
	BagClear = FALSE
ENDIF

;Step 4 - Bag full wait for operator to open
IF (STEP = 4) THEN
	O_BagReady = TRUE
	;O_OpenCatch = TRUE
	IF I_OpenBag THEN
		D[924] = 5
	ENDIF
ENDIF

;Step 5 - Open bag
TON_10ms((STEP = 5),600,MinOpen,MinOpenET)
IF (STEP = 5) THEN
	O_OpenBag 	= TRUE
	O_OpenCatch = TRUE
	IF  MinOpen THEN
		D[924] = 6
	ENDIF
ENDIF

;Step 6 - Open bag wait for operator to confirm empty
IF (STEP = 6) THEN
	O_BagReady 	= Std.Clock1s
	O_OpenBag 	= TRUE
	O_OpenCatch = TRUE
	IF I_OpenBag THEN
		D[924] = 7
	ENDIF
ENDIF

;Step 7 - Close bag
TON_10ms((STEP = 7),500,CloserDown,CloserDownET)
IF (STEP = 7) THEN
	O_OpenCatch = TRUE
	IF CloserDown THEN
		D[924] = 1
	ENDIF
ENDIF

;Alarms
TimerAlarm.IN 		= NOT PLS AND (Alarm[mySeq].Name > 0)
TimerAlarm.PT 		= Alarm[mySeq].Time
TimerAlarm FUB TON_10ms()
Alarm[mySeq].On 	= TimerAlarm.Q
Alarm[mySeq].ET 	= TimerAlarm.ET

;PLC Outputs
;-----------
Y[5].Y05	= O_BagReady
Y[7].Y14	= O_OpenCatch
Y[7].Y15 	= O_OpenBag

END_PROGRAM
```

#### 7_svc1.var
```iecst
VAR RETAIN
	STEP : UINT;
END_VAR
VAR
	PLS : BOOL;
END_VAR
VAR RETAIN
	LASTSTEP : UINT;
END_VAR
VAR
	I_CarrAtTop : BOOL;
	I_BagOnCarr : BOOL;
	I_CarrAtBottom : BOOL;
	O_OpenCarrStop : BOOL;
	O_MoveCarrDown : BOOL;
	O_MoveCarrUp : BOOL;
	BagSettled : BOOL;
	O_OpenBufferStop : BOOL;
	BagAtBuffer : BOOL;
	MoveUpToFullOut : BOOL;
	MoveDownToBot : BOOL;
	Status : UINT;
	HighSpeedDoneET : TIME;
	I_BagBagReleased : BOOL;
	TONHighSpeed : TON_10ms;
	TimerAlarm : TON_10ms;
	HighSpeedTime : UINT;
	HighSpeedDone : BOOL;
	BagAtBufferET : TIME;
	I_BagAtBufferStop : BOOL;
	MoveDownEBagIn : BOOL;
	DDDDDD : BOOL;
	BagSettledET : TIME;
	I_CarriageAtTop : BOOL;
	I_CarriageAtBottom : BOOL;
	I_BagOnCarriage : BOOL;
	I_BagReleased : BOOL;
	O_MoveUp : BOOL;
	O_MoveDown : BOOL;
	O_OpenStop : BOOL;
	SettledOnCarriage : BOOL;
	SettledOnCarriageET : UDINT;
	E : BOOL;
	HighSpeedUp : BOOL;
	HighSpeedUpET : UDINT;
	HighSpeedDn : BOOL;
	HighSpeedDnET : UDINT;
	I_OpenBag : BOOL;
	I_DischBagOpened : BOOL;
	O_BagReady : BOOL;
	O_OpenCatch : BOOL;
	O_OpenBag : BOOL;
	O_CloseBag : BOOL;
	TopBagOpen : BOOL;
	TopBagOpenET : UDINT;
	OpenCatch : BOOL;
	BagClear : BOOL;
	MinOpen : BOOL;
	MinOpenET : UDINT;
	CloserDown : BOOL;
	CloserDownET : UDINT;
	mySeq : INT;
END_VAR
```

### Program Logical/Sequences/10ms/25_cp16 (IEC, version 1.00.0) - * SBSN1 Bagstacker Ongoing 

#### 10_bsonCyclic.ab
```automation-basic
PROGRAM _CYCLIC
(* cyclic program *)

;----------------------------------------
;Sequence 14 - Ongoing Bag Stacker D[910]
;----------------------------------------

;Inputs
I_BagatBuffer       = X[2].X10

O_Reset = FALSE
O_OpenBuffer = FALSE
O_SelectLine13_1 = FALSE
O_SelectLine14_1 = FALSE
O_SelectLine15_1 = FALSE
O_SelectLine16_1 = FALSE
O_SelectLine16_2 = FALSE

mySeq				= 25	;Sequence number

Alarm[mySeq].Name 	= 0
Alarm[mySeq].Bag	= 54
Alarm[mySeq].Beacon	= TRUE
Alarm[mySeq].Extra	= 0
Alarm[mySeq].Time	= 3000
;Setup Sequence
;-----------------------
STEP = D[925]

;Setup Pulse contact
PLS = (STEP <> LASTSTEP)
LASTSTEP = STEP

;Alarm
;TON_10ms(((NOT PLS) AND ((STEP = 3) OR (STEP = 4) OR (STEP = 8))),6000,Alarm[10],AlarmET[10])

IF (STEP = 0) THEN
	;Do Nothing
ENDIF

;Reset Points
TON_10ms((STEP = 1),250,Reset,ResetET)
IF (STEP = 1) THEN
	O_Reset = TRUE

    Destination = 0
	IF Reset THEN
		D[925] = 2
	ENDIF
ENDIF

;Wait for bag at buffer stop
TON_10ms(I_BagatBuffer,300,BagSettledBuffer,BagSettledBufferET)
IF (STEP = 2) THEN
	;Allocate Destination to Bag
	IF (Bag[54].Dst > 0) AND (Bag[54].Cat > 0) THEN
		Destination = Bag[54].Dst
	ENDIF
	IF (Bag[54].Dst = 0)AND (Bag[54].Cat > 0) THEN
		IF (Line[D[3000+Bag[54].Cat]].SpaceBIT>0) AND (D[D[3000+Bag[54].Cat] +10] > 0)    THEN
			Bag[54].Dst = USINT(D[3000+Bag[54].Cat])
		ELSE IF (Line[D[3100+Bag[54].Cat]].SpaceBIT>0) AND (D[D[3100+Bag[54].Cat] +10] > 0)THEN
			Bag[54].Dst = USINT(D[3100+Bag[54].Cat])
		ENDIF
	ENDIF
		IF ((BagSettledBuffer) AND (Bag[54].Cat > 0) AND (Bag[54].Dst > 0))THEN

			D[925] = 3
		ENDIF
	//ENDIF
ENDIF

;Enable requesting discharger to send a bag
IF (STEP = 3) THEN
	IF (Bag[54].Dst = 7) THEN
		IF ((Bag[66].Cat = 0) AND (Line[7].Clear)) THEN
            C[7] 	= 0

			D[925] 	= 4
		ENDIF
	ELSE IF ((Bag[54].Dst > 0) AND (Bag[54].Dst <= 8) AND (Bag[54].Dst <> 7)) THEN
		IF ((Bag[52].Cat = 0) AND (Line[16].Clear)) THEN
            C[16] 	= 0
            D[40]	= 1
			D[925] 	= 5
		ENDIF
	ENDIF
ENDIF

;Send bag to CDC7 Line
IF (STEP = 4) THEN
	//IF (D[40] = 2) THEN
		O_OpenBuffer = TRUE
        O_SelectLine16_2 = TRUE
		IF (Line[7].Full) THEN
			IF (Bag[54].Cat>0) AND (Bag[66].Cat=0) THEN
				Bag[66] = Bag[54]
				Bag[54] = Bag[0]
				Bag[66].Dst = 0
			ENDIF
        // E[329] = 0	;Clear Dest
		//	BAGMOVE2(TRUE,mem_adr_E,54,66,BagSpacing)
         Line[7].SpaceBIT = (Line[7].SpaceBIT - 1)
		D[925] = 1
		ENDIF
	Alarm[mySeq].Name = almBagNotReleased
ENDIF

;Send bag to CP13 Line
IF (STEP = 5) THEN
	//IF (D[40] = 1) THEN
		O_OpenBuffer = TRUE
		IF (Line[16].Full) THEN
		//	BAGMOVE2(TRUE,mem_adr_E,54,52,BagSpacing)
			IF (Bag[54].Cat>0) AND (Bag[52].Cat=0) THEN
				Bag[52] = Bag[54]
				Bag[54] = Bag[0]
			ENDIF
		D[925] = 1
		ENDIF
	Alarm[mySeq].Name =  almBagNotReleased
ENDIF
;Alarms
TimerAlarm.IN 		= NOT PLS AND (Alarm[mySeq].Name > 0)
TimerAlarm.PT 		= Alarm[mySeq].Time
TimerAlarm FUB TON_10ms()
Alarm[mySeq].On 	= TimerAlarm.Q
Alarm[mySeq].ET 	= TimerAlarm.ET

Y[7].Y11 = O_Reset

Y[2].Y10 = O_OpenBuffer
Y[7].Y10 = O_SelectLine16_2

END_PROGRAM
```

#### 10_bson.var
```iecst
VAR
	I_OnLineA : BOOL;
	I_TiltA : BOOL;
	I_TiltB : BOOL;
	I_Bagout : BOOL;
	O_OpenBufferStop : BOOL;
	O_SelectLineA : BOOL;
	O_SelectLineB : BOOL;
	O_OpenStops : BOOL;
	O_TiltCylinder : BOOL;
	O_OperatePusher : BOOL;
	PLS : BOOL;
END_VAR
VAR RETAIN
	LASTSTEP : UINT;
	STEP : UINT;
END_VAR
VAR
	TiltDownET : UDINT;
	TiltDown : BOOL;
	TiltUpET : UDINT;
	TiltUp : BOOL;
	NotFullET : UDINT;
	NotFull : BOOL;
	RequirePusherET : UDINT;
	Pushed : BOOL;
	PushedET : UDINT;
	BagAtTiltET : TIME;
	BagAtTilt : BOOL;
	PointReset : BOOL;
	PointResetET : TIME;
	TimerAlarm : TON_10ms;
	ResetPoint : BOOL;
	ResetPointET : UDINT;
	BagatTilt : BOOL;
	BagatTiltET : UDINT;
	I_BagatBuffer : BOOL;
	O_Reset : BOOL;
	O_OpenBuffer : BOOL;
	O_SelectLine13_1 : BOOL;
	O_SelectLine14_1 : BOOL;
	O_SelectLine15_1 : BOOL;
	O_SelectLine16_1 : BOOL;
	O_SelectLine16_2 : BOOL;
	mySeq : INT;
	Reset : BOOL;
	ResetET : UDINT;
	Destination : INT;
	BagSettledBuffer : BOOL;
	BagSettledBufferET : UDINT;
END_VAR
```

### Program Logical/Sequences/10ms/26_cic8 (IEC) - * SBSF1 Bagstacker Offgoing

#### 11_bsoff.var
```iecst
VAR RETAIN
	STEP : UINT;
END_VAR
VAR
	PLS : BOOL;
END_VAR
VAR RETAIN
	LASTSTEP : UINT;
END_VAR
VAR
	LevellerDownET : TIME;
	O_LevelCylinder : BOOL;
	O_SelectLineB : BOOL;
	O_SelectLineA : BOOL;
	I_OutLineB : BOOL;
	LevellerDown : BOOL;
	LevellerUp : BOOL;
	LevellerUpET : TIME;
	I_TiltB : BOOL; (* SPR1 Trolley past stop *)
	I_OutLineA : BOOL;
	O_OpenRockSep : BOOL;
	O_OpenLineAStop : BOOL;
	O_OpenLineBStop : BOOL;
	I_RockSepA : BOOL;
	I_RockSepB : BOOL;
	I_TiltA : BOOL; (* SBS1 ON Bag on stacker *)
	O_LevelCylinderUP : BOOL;
	PRLineClearET : ARRAY[0..4] OF TIME;
	SettledLevel : BOOL;
	SettledLevelET : TIME;
	SettledInSepsET : TIME;
	SettledInSeps : BOOL;
	LevelClearET : TIME;
	LevelClear : BOOL;
	TimerAlarm : TON_10ms;
	I_LevelA : BOOL;
	I_LevelB : BOOL;
	I_AtRotary : BOOL;
	O_RotatePoint : BOOL;
	O_OpenRotaryPoint : BOOL;
	AlarmET : UDINT;
	SelectA : BOOL;
	SelectAET : UDINT;
	RockerReady : BOOL;
	RockerReadyET : UDINT;
	LevellerFull : BOOL;
	LevellerFullET : UDINT;
	SettledInRotary : BOOL;
	SettledInRotaryET : UDINT;
	PointRotated : BOOL;
	PointRotatedET : UDINT;
	I_PaddleinPosition : BOOL;
	I_BaginIncline : BOOL;
	I_BagOut : BOOL;
	O_RunMotor : BOOL;
	O_Reset : BOOL;
	Reset : BOOL;
	ResetET : UDINT;
	BagSettled : BOOL;
	BagSettledET : UDINT;
	BagInIncline : BOOL;
	NearTop : BOOL;
	NearTopET : UDINT;
	RanOn : BOOL;
	RanOnET : UDINT;
	MySeq : INT;
END_VAR
```

#### 11_bsoffCyclic.ab
```automation-basic
PROGRAM _CYCLIC
  	(* cyclic program *)

;-----------------------------------------
;Sequence 11 - Offgoing Bag Stacker D[911]
;-----------------------------------------

;Inputs
I_PaddleinPosition	= X[2].X07
I_BaginIncline		= X[2].X06
I_BagOut            = X[2].X08

MySeq                   = 26
O_RunMotor 			= FALSE
O_Reset             = FALSE
Request.CIC[8] = FALSE
Enable.CDC[5]   = FALSE
Enable.CDC[6]   = FALSE

;O_SelectLineA			= FALSE
;O_SelectLineB			= FALSE
O_RotatePoint			= FALSE
O_OpenRockSep			= FALSE
O_OpenLineAStop			= FALSE
O_OpenLineBStop			= FALSE
O_LevelCylinder			= FALSE
O_OpenRotaryPoint		= FALSE

Alarm[MySeq].Name 			= 0 ;Clear sequence alarm name
Alarm[MySeq].Bag 			= 0
Alarm[MySeq].Beacon			= TRUE
Alarm[MySeq].Extra			= 0
Alarm[MySeq].Time			= 3000

;Setup Sequence
;-----------------------
STEP = D[926]
;Setup Pulse contact
PLS = (STEP <> LASTSTEP)
LASTSTEP = STEP

;Alarm
;TON_10ms(((NOT PLS) AND ((STEP = 3) OR (STEP = 7) OR (STEP = 8) OR (STEP = 9))),3000,Alarm[11],AlarmET[11])

;Select Line 'A'
TON_10ms(((STEP = 1)),200,Reset,ResetET)
IF (STEP = 1) THEN
	O_RunMotor = (NOT I_PaddleinPosition)
	O_Reset = TRUE

	IF I_PaddleinPosition AND Reset THEN
		D[926] = 2
	ENDIF
	Alarm[MySeq].Name 			= almSwitchFault
ENDIF

;Check incline clear
IF (STEP = 2) THEN
	IF NOT (I_BaginIncline) THEN
		D[926] = 3
	ENDIF
ENDIF

;Check request release from CIC7 - CDC5 - CDC6
IF (STEP = 3) THEN
	IF (Request.CIC[7]) THEN ;Request release from CIC7
		D[51] = 1
		IF (D[51] > 0) THEN
			D[926] = 4
		ENDIF
	ELSE IF (Request.CDC[6]) THEN ;Request release from CDC5
        D[51] = 2
		IF (D[51] > 0) THEN
			D[926] = 4
		ENDIF
	ELSE IF (Request.CDC[5]) THEN ;Request release from CDC6
        D[51] = 3
		IF (D[51] > 0) THEN
			D[926] = 4
		ENDIF
	ENDIF
ENDIF

;Let bag settle at base of incline
TON_10ms((STEP = 4) AND I_BaginIncline,400,BagSettled,BagSettledET)
IF (STEP = 4) THEN
	IF I_BaginIncline THEN
		BagInIncline = TRUE
	ENDIF
	Enable.CIC[7] = (D[51] = 1)
    Enable.CDC[6] = (D[51] = 2)
    Enable.CDC[5] = (D[51] = 3)
	IF (BagSettled) THEN
		D[51]        = 0
		D[926] = 5
	ENDIF
	Alarm[MySeq].Name 			= almSwitchFault
	ELSE
	BagInIncline = FALSE

ENDIF

;Move bag up incline to save time
TON_10ms((STEP = 5),500,NearTop,NearTopET)
IF (STEP = 5) THEN
	O_RunMotor = TRUE
	IF ((NearTop) AND NOT (Enable.CIC[1])) THEN
		D[926] = 6
	ENDIF
ENDIF

;Check Destination Of Bag
TON_10ms((STEP = 6),30,RanOn,RanOnET)
IF (STEP = 6) THEN
	O_RunMotor = NOT RanOn
	  Request.CIC[8] = TRUE
	IF (Enable.CIC[8]) THEN
		D[926]  = 7
	ENDIF
ENDIF

;Run incline conveyor until bag at destination
IF (STEP = 7) THEN
	O_RunMotor = TRUE
	IF (I_BagOut) THEN
		D[926] = 1
	ENDIF
	Alarm[MySeq].Name 			= almSwitchFault
ENDIF

;Alarms
TimerAlarm.IN 	= NOT PLS AND (Alarm[MySeq].Name > 0)
TimerAlarm.PT 	= Alarm[MySeq].Time
TimerAlarm FUB TON_10ms()
Alarm[MySeq].On 	= TimerAlarm.Q
Alarm[MySeq].ET 	= TimerAlarm.ET

;Y000 = O_SelectLineA
;Y000 = O_SelectLineB
Y[2].Y16 = O_RunMotor

Y[8].Y15 = O_Reset

END_PROGRAM
```

### Program Logical/Sequences/10ms/27_csb2 (IEC, version 1.00.0) - * SVC2 2-level - Inverter

#### 12_svc2Cyclic.ab
```automation-basic
PROGRAM _CYCLIC
	(* cyclic program *)

;--------------------------------------------
;Sequence 8 - SVC1 Vertical conveyor 1 D[908]
;--------------------------------------------

;Inputs
I_OpenBag				= X[2].X12

I_DischBagOpened		= (D[909] = 7)

mySeq                   = 27
O_BagReady				= FALSE
O_OpenCatch				= FALSE
O_OpenBag				= FALSE
O_CloseBag				= FALSE

Enable.CDC4Open		    = FALSE

;Alarm[mySeq].Name 	= 0
Alarm[mySeq].Bag	= 58
Alarm[mySeq].Beacon	= TRUE
Alarm[mySeq].Extra	= 0
Alarm[mySeq].Time	= 3000
;Setup Sequence
;-----------------------
STEP = D[927]
;Setup Pulse contact
PLS = (STEP <> LASTSTEP)
LASTSTEP = STEP

;Alarm
;TON_10ms(((NOT PLS) AND ((STEP = 2) OR (STEP = 3) OR (STEP = 6))),3000,Alarm[12],AlarmET[12])

;Step 1 - Check signals
IF (STEP = 1) THEN
	IF (NOT I_OpenBag) THEN
		D[927] = 2
	ENDIF
ENDIF

;Step 2 - Enable discharger to open
TON_10ms(I_DischBagOpened,600,TopBagOpen,TopBagOpenET)
IF (STEP = 2) THEN
	Enable.CDC4Open = I_OpenBag
	O_BagReady = (D[909] = 5)
	IF I_OpenBag THEN
		OpenCatch = TRUE
	ENDIF
	O_OpenCatch = OpenCatch
	IF TopBagOpen THEN
		D[927] 		= 3
	ENDIF
	ELSE
	OpenCatch = FALSE
ENDIF

;Step 3 - Bag being loaded
IF (STEP = 3) THEN
		O_BagReady = Std.Clock500ms
		O_OpenCatch = TRUE
		IF I_OpenBag THEN
			BagClear = TRUE
		ENDIF
		IF BagClear AND NOT I_OpenBag THEN
			D[927] = 4
		ENDIF
	ELSE
	BagClear = FALSE
ENDIF

;Step 4 - Bag full wait for operator to open
IF (STEP = 4) THEN
	O_BagReady = TRUE
	;O_OpenCatch = TRUE
	IF I_OpenBag THEN
		D[927] = 5
	ENDIF
ENDIF

;Step 5 - Open bag
TON_10ms((STEP = 5),600,MinOpen,MinOpenET)
IF (STEP = 5) THEN
	O_OpenBag 	= TRUE
	O_OpenCatch = TRUE
	IF  MinOpen THEN
		D[927] = 6
	ENDIF
ENDIF

;Step 6 - Open bag wait for operator to confirm empty
IF (STEP = 6) THEN
	O_BagReady 	= Std.Clock500ms
	O_OpenBag 	= TRUE
	O_OpenCatch = TRUE
	IF I_OpenBag THEN
		D[927] = 7
	ENDIF
ENDIF

;Step 7 - Close bag
TON_10ms((STEP = 7),500,CloserDown,CloserDownET)
IF (STEP = 7) THEN
	O_OpenCatch = TRUE
	IF CloserDown THEN
		D[927] = 1
	ENDIF
ENDIF

;Alarms
TimerAlarm.IN 		= NOT PLS AND (Alarm[mySeq].Name > 0)
TimerAlarm.PT 		= Alarm[mySeq].Time
TimerAlarm FUB TON_10ms()
Alarm[mySeq].On 	= TimerAlarm.Q
Alarm[mySeq].ET 	= TimerAlarm.ET

;Outputs
Y[2].Y07	= O_BagReady
Y[2].Y05	= O_OpenCatch
Y[2].Y06 	= O_OpenBag

END_PROGRAM
```

#### 12_svc2.var
```iecst
VAR
	I_CarrAtTop : BOOL;
	I_CarrAtBottom : BOOL;
END_VAR
VAR RETAIN
	STEP : UINT;
END_VAR
VAR
	PLS : BOOL;
END_VAR
VAR RETAIN
	LASTSTEP : UINT;
END_VAR
VAR
	O_MoveCarrUp : BOOL;
	O_OpenCarrStop : BOOL;
	O_MoveCarrDown : BOOL;
	I_BagOnCarr : BOOL;
	Speed1 : BOOL;
	MoveDownToBot : BOOL;
	Speed2 : BOOL;
	O_SelectSP1 : BOOL;
	MoveUpToFullOut : BOOL;
	I_BagReleased : BOOL;
	TimerAlarm : TON_10ms;
	I_CarrAtEBagOut : BOOL;
	O_SelectPoint : BOOL;
	O_OpenFullBuffer : BOOL;
	HighSpeedDone : BOOL;
	HighSpeedTime : UDINT;
	TONHighSpeed : TON_10ms;
	MoveDownEBagIn : BOOL;
	HighSpeedDoneET : TIME;
	SettledAtBuffer : BOOL;
	SettledAtBufferET : TIME;
	I_CarriageAtTop : BOOL;
	I_CarriageAtBottom : BOOL;
	I_BagOnCarriage : BOOL;
	I_BagAtBuffer : BOOL;
	O_MoveUp : BOOL;
	O_MoveDown : BOOL;
	O_OpenStop : BOOL;
	O_OpenBufferStop : BOOL;
	EBagReady : BOOL;
	EBagReadyET : UDINT;
	BagSettled : BOOL;
	BagSettledET : UDINT;
	HighSpeedUp : BOOL;
	HighSpeedUpET : UDINT;
	HighSpeedDn : BOOL;
	HighSpeedDnET : UDINT;
	I_OpenBag : BOOL;
	I_DischBagOpened : BOOL;
	O_BagReady : BOOL;
	O_OpenCatch : BOOL;
	O_OpenBag : BOOL;
	O_CloseBag : BOOL;
	TopBagOpen : BOOL;
	TopBagOpenET : UDINT;
	OpenCatch : BOOL;
	BagClear : BOOL;
	MinOpen : BOOL;
	MinOpenET : UDINT;
	CloserDown : BOOL;
	CloserDownET : UDINT;
	mySeq : INT;
END_VAR
```

### Program Logical/Sequences/10ms/zzAI2744 (IEC) - Weight 

#### zzAI2744Cyclic.ab - Cyclic code
```automation-basic
(********************************************************************
 * COPYRIGHT -- Kannegiesser UK Ltd
 ********************************************************************
 * Program: zzAI2744
 * File: zzAI2744Cyclic.ab
 * Author: zmclaren
 * Created: May 25, 2012
 ********************************************************************
 * Implementation of program zzAI2744
 ********************************************************************)

PROGRAM _CYCLIC
(* First we need to see if the last value is different to the previous one, *)
(* Then we will set the counters for each to zero *)
(* Also the Config Outputs will need setting to 0*)
IF (D[998] = 0) THEN
	LOOP i = 1 TO 54 DO
		IF (LastRawValue[i] = AI261Raw[i])THEN        (* We have no change between the  two values *)
			IF (NoChangeCounter[i] >= 21) THEN          (* We need to reset the output back to zero *)
				ConfigOutput[i]    = 0
			ELSE
				IF (NoChangeCounter[i] = 20) THEN  (* We have had 20 cycles with no change on the input *)
					NoChangeCounter[i] = NoChangeCounter[i] + 1
					ConfigOutput[i]    = %00110001  (* Make a change to both the Data Rate and teh Range *)
				ELSE
					NoChangeCounter[i] = NoChangeCounter[i] + 1  (* Increment the no change counter *)
				ENDIF
			ENDIF
		ELSE     (* There has been a change between the two  Values so store the old value and clear the counter *)
			LastRawValue[i] = AI261Raw[i]  (* Store the Last Value *)
			NoChangeCounter[i] = 0         (* Reset the Counter *)
			ConfigOutput[i]    = 0         (* Leave the configuration as  0 *)
		ENDIF
	ENDLOOP
ENDIF

END_PROGRAM
```

### Program Logical/Sequences/10ms/ssr (IEC) - *Speed Reducers

#### p.var
```iecst
VAR
	myHaltSys : BOOL;
	O_CloseBrush : ARRAY[0..5] OF BOOL;
	I_BagApproach : ARRAY[0..5] OF BOOL;
	TON_OpenBrush : ARRAY[0..5] OF TON_10ms;
	n : USINT;
	myZone : INT;
	SettledAtSep : BOOL;
	O_OpenSep : BOOL;
	CloseSep : BOOL;
	I_BagAtRollerRockerBeforePDS1 : BOOL;
	SettledAtSepET : UDINT;
	CloseSepET : UDINT;
	I_BagAtBottom : BOOL;
	PR3_LineClear : BOOL;
	PR3_LineClearET : UDINT;
	PR4_LineClear : BOOL;
	PR4_LineClearET : UDINT;
END_VAR
```

#### p.ab
```automation-basic
;-------------
;Speed Reducer
;-------------

PROGRAM _INIT

END_PROGRAM
PROGRAM _CYCLIC

;Empty bag pressure relief CPR2
TON_10ms((Line[13].Clear AND X[7].X07 AND NOT Y[7].Y07),500,PR3_LineClear,PR3_LineClearET)
IF PR3_LineClear THEN
	C[13] 	= 0
	Y[7].Y07 	= TRUE
ENDIF
IF Line[13].Full THEN
	Y[7].Y07 	= FALSE
ENDIF

;Full bag pressure relief CPR3 - Line 5
TON_10ms((Line[6].Clear AND X[7].X09 AND NOT Y[7].Y09),500,PR4_LineClear,PR4_LineClearET)
IF PR4_LineClear THEN
	C[6] 	= 0
	Y[7].Y09 	= TRUE
ENDIF
IF Line[6].Full THEN
	IF (Bag[26].Cat>0) AND (Bag[66].Cat=0) THEN
		;		Bag[66] = Bag[26]
		;		Bag[26] = Bag[0]
			ENDIF
//	BAGMOVE2(Y[7].Y09,mem_adr_E,26,66,BagSpacing)
;	Y[7].Y09 	= FALSE
ENDIF

END_PROGRAM
```

- Program Logical/Sequences/10ms/zzIndi (IEC) - * Indication pictures on graphics (no source held here)

- Program Logical/Sequences/10ms/zzTCPIP (IEC, version 5.00.0) - * TCP IP Communications For Driver V5.0 and above (no source held here)

### Program Logical/Sequences/10ms/zzForceO (IEC) - * PLC Output forcing from graphics

#### zzforceo.var
```iecst
VAR
	YForce : CardOutputs;
	YForceVal : CardOutputs;
	Force : UINT := 0;
	n : UINT;
	myForceState : UINT;
	myForceCard : UINT;
	myForceValue : UINT;
END_VAR
```

#### zzforceo.ab
```automation-basic
;----------------------------
;Output forcing from Graphics
;----------------------------

;Version 1.00 02/09/2006 D.J. First Issue
;Version 2.00 20/11/2009 D.J. Changed to 8 I/O inputs per card

PROGRAM _INIT

;Clear force registers

D[380] = 0
D[381] = 0
D[382] = 0
D[383] = 0
D[384] = 0
D[385] = 0
D[386] = 0
D[386] = 0
D[387] = 0
D[388] = 0
D[389] = 0
D[390] = 0
D[391] = 0
D[392] = 0
D[393] = 0
D[394] = 0
D[395] = 0
D[396] = 0
D[396] = 0
D[397] = 0
D[398] = 0
D[399] = 0

;Clear force disable
memset(ADR(YForceDisable),0, SIZEOF(YForceDisable))

END_PROGRAM

PROGRAM _CYCLIC

LOOP Force = 1 TO 4 DO

	n = ((Force - 1) * 5)

	myForceCard 	= D[380 + n]
	myForceState 	= D[383 + n]
	myForceValue 	= D[384 + n]

	IF (myForceCard > Std.MaxIO) THEN
		myForceCard = 0
	ENDIF

	YForce.Y01 		= BIT_TST(myForceState,0)
	YForce.Y02 		= BIT_TST(myForceState,1)
	YForce.Y03 		= BIT_TST(myForceState,2)
	YForce.Y04 		= BIT_TST(myForceState,3)
	YForce.Y05 		= BIT_TST(myForceState,4)
	YForce.Y06 		= BIT_TST(myForceState,5)
	YForce.Y07 		= BIT_TST(myForceState,6)
	YForce.Y08 		= BIT_TST(myForceState,7)

	YForceVal.Y01 	= BIT_TST(myForceValue,0)
	YForceVal.Y02 	= BIT_TST(myForceValue,1)
	YForceVal.Y03 	= BIT_TST(myForceValue,2)
	YForceVal.Y04 	= BIT_TST(myForceValue,3)
	YForceVal.Y05 	= BIT_TST(myForceValue,4)
	YForceVal.Y06 	= BIT_TST(myForceValue,5)
	YForceVal.Y07 	= BIT_TST(myForceValue,6)
	YForceVal.Y08 	= BIT_TST(myForceValue,7)

	Y[myForceCard].Y01 = (Y[myForceCard].Y01 AND NOT YForce.Y01) OR (YForce.Y01 AND YForceVal.Y01 AND NOT YForceDisable[myForceCard].Y01)
	Y[myForceCard].Y02 = (Y[myForceCard].Y02 AND NOT YForce.Y02) OR (YForce.Y02 AND YForceVal.Y02 AND NOT YForceDisable[myForceCard].Y02)
	Y[myForceCard].Y03 = (Y[myForceCard].Y03 AND NOT YForce.Y03) OR (YForce.Y03 AND YForceVal.Y03 AND NOT YForceDisable[myForceCard].Y03)
	Y[myForceCard].Y04 = (Y[myForceCard].Y04 AND NOT YForce.Y04) OR (YForce.Y04 AND YForceVal.Y04 AND NOT YForceDisable[myForceCard].Y04)
	Y[myForceCard].Y05 = (Y[myForceCard].Y05 AND NOT YForce.Y05) OR (YForce.Y05 AND YForceVal.Y05 AND NOT YForceDisable[myForceCard].Y05)
	Y[myForceCard].Y06 = (Y[myForceCard].Y06 AND NOT YForce.Y06) OR (YForce.Y06 AND YForceVal.Y06 AND NOT YForceDisable[myForceCard].Y06)
	Y[myForceCard].Y07 = (Y[myForceCard].Y07 AND NOT YForce.Y07) OR (YForce.Y07 AND YForceVal.Y07 AND NOT YForceDisable[myForceCard].Y07)
	Y[myForceCard].Y08 = (Y[myForceCard].Y08 AND NOT YForce.Y08) OR (YForce.Y08 AND YForceVal.Y08 AND NOT YForceDisable[myForceCard].Y08)

ENDLOOP

END_PROGRAM
```

### Program Logical/Sequences/10ms/zzIO (IEC) - * PLC Inputs and Outputs to Graphics

#### zzio.ab
```automation-basic
PROGRAM _CYCLIC
(* cyclic program *)

;Transmit I/O to PC Graphics

;-----------------------------------------------------------------------------------------
;Version 1.00 19/12/2005 D.J. First Issue
;Version 2.00 13/11/2006 D.J. All I/O Sent to Graphics
;Version 3.00 02/05/2007 D.J. Do more than 1 card per scan
;Version 4.00 20/11/2009 D.J. Changed from 16 I/O to 8 I/O Per Card (2 cards per 16-bit D)
;-----------------------------------------------------------------------------------------

LOOP n = 1 TO 5 DO ;Do 5 * 2 cards per scan

	CurrentCard 	= CurrentCard + 2
	DataRegister 	= DataRegister + 1

	IF (CurrentCard > Std.MaxIO) OR (DataRegister > 199) THEN
		CurrentCard = 0
		DataRegister = 0
	ENDIF

	InputCard.Input[0] 	= X[CurrentCard + 0].X01
	InputCard.Input[1] 	= X[CurrentCard + 0].X02
	InputCard.Input[2] 	= X[CurrentCard + 0].X03
	InputCard.Input[3] 	= X[CurrentCard + 0].X04
	InputCard.Input[4] 	= X[CurrentCard + 0].X05
	InputCard.Input[5] 	= X[CurrentCard + 0].X06
	InputCard.Input[6] 	= X[CurrentCard + 0].X07
	InputCard.Input[7] 	= X[CurrentCard + 0].X08
	InputCard.Input[8] 	= X[CurrentCard + 1].X01
	InputCard.Input[9] 	= X[CurrentCard + 1].X02
	InputCard.Input[10] = X[CurrentCard + 1].X03
	InputCard.Input[11] = X[CurrentCard + 1].X04
	InputCard.Input[12] = X[CurrentCard + 1].X05
	InputCard.Input[13] = X[CurrentCard + 1].X06
	InputCard.Input[14] = X[CurrentCard + 1].X07
	InputCard.Input[15] = X[CurrentCard + 1].X08
	InputCard FUB BIT_ENCODE()

	D[400 + DataRegister] 	= InputCard.Output

	OutputCard.Input[0] 	= Y[CurrentCard + 0].Y01
	OutputCard.Input[1] 	= Y[CurrentCard + 0].Y02
	OutputCard.Input[2] 	= Y[CurrentCard + 0].Y03
	OutputCard.Input[3] 	= Y[CurrentCard + 0].Y04
	OutputCard.Input[4] 	= Y[CurrentCard + 0].Y05
	OutputCard.Input[5] 	= Y[CurrentCard + 0].Y06
	OutputCard.Input[6] 	= Y[CurrentCard + 0].Y07
	OutputCard.Input[7] 	= Y[CurrentCard + 0].Y08
	OutputCard.Input[8] 	= Y[CurrentCard + 1].Y01
	OutputCard.Input[9] 	= Y[CurrentCard + 1].Y02
	OutputCard.Input[10] 	= Y[CurrentCard + 1].Y03
	OutputCard.Input[11] 	= Y[CurrentCard + 1].Y04
	OutputCard.Input[12] 	= Y[CurrentCard + 1].Y05
	OutputCard.Input[13] 	= Y[CurrentCard + 1].Y06
	OutputCard.Input[14] 	= Y[CurrentCard + 1].Y07
	OutputCard.Input[15] 	= Y[CurrentCard + 1].Y08
	OutputCard FUB BIT_ENCODE()

	D[600 + DataRegister] 	= OutputCard.Output

ENDLOOP
END_PROGRAM
```

### Program Logical/Sequences/10ms/zzOk (IEC) - * PLC Status to Graphics

#### zzok.var
```iecst
VAR
	n : UINT;
	Module : UINT;
	ModuleEncode : BIT_ENCODE;
	StnModuleEncode : BIT_ENCODE;
	StnModule : UINT;
END_VAR
```

#### zzok.ab
```automation-basic
PROGRAM _CYCLIC
(* cyclic program *)

;Transmit I/O Status to PC Graphics up-to 400 I/O Modules

;----------------------------------------
;Version 1.00 10/12/2007 D.J. First Issue
;----------------------------------------

Module = Module + 1

IF (Module > 24) THEN
	Module = 0
ENDIF

n = (Module * 16)

ModuleEncode.Input[0] 	= OK[n + 1]
ModuleEncode.Input[1] 	= OK[n + 2]
ModuleEncode.Input[2] 	= OK[n + 3]
ModuleEncode.Input[3] 	= OK[n + 4]
ModuleEncode.Input[4] 	= OK[n + 5]
ModuleEncode.Input[5] 	= OK[n + 6]
ModuleEncode.Input[6] 	= OK[n + 7]
ModuleEncode.Input[7] 	= OK[n + 8]
ModuleEncode.Input[8] 	= OK[n + 9]
ModuleEncode.Input[9] 	= OK[n + 10]
ModuleEncode.Input[10] 	= OK[n + 11]
ModuleEncode.Input[11] 	= OK[n + 12]
ModuleEncode.Input[12] 	= OK[n + 13]
ModuleEncode.Input[13] 	= OK[n + 14]
ModuleEncode.Input[14] 	= OK[n + 15]
ModuleEncode.Input[15] 	= OK[n + 16]
ModuleEncode FUB BIT_ENCODE()

D[320 + Module] 	= ModuleEncode.Output

StnModule = StnModule + 1

IF (StnModule > 7) THEN
	StnModule = 0
ENDIF

n = (StnModule * 16)

StnModuleEncode.Input[0] 	= StnOK[n + 1]
StnModuleEncode.Input[1] 	= StnOK[n + 2]
StnModuleEncode.Input[2] 	= StnOK[n + 3]
StnModuleEncode.Input[3] 	= StnOK[n + 4]
StnModuleEncode.Input[4] 	= StnOK[n + 5]
StnModuleEncode.Input[5] 	= StnOK[n + 6]
StnModuleEncode.Input[6] 	= StnOK[n + 7]
StnModuleEncode.Input[7] 	= StnOK[n + 8]
StnModuleEncode.Input[8] 	= StnOK[n + 9]
StnModuleEncode.Input[9] 	= StnOK[n + 10]
StnModuleEncode.Input[10] 	= StnOK[n + 11]
StnModuleEncode.Input[11] 	= StnOK[n + 12]
StnModuleEncode.Input[12] 	= StnOK[n + 13]
StnModuleEncode.Input[13] 	= StnOK[n + 14]
StnModuleEncode.Input[14] 	= StnOK[n + 15]
StnModuleEncode.Input[15] 	= StnOK[n + 16]
StnModuleEncode FUB BIT_ENCODE()

D[350 + StnModule] 	= StnModuleEncode.Output
END_PROGRAM
```

### udp_CTT.typ
```iecst
TYPE
 RX_Buffer_CCT_PLC :  STRUCT
  UpLeft : USINT;
  DwnLeft : USINT;
  UpRight : USINT;
  DwnRight : USINT;
  sendRequest : USINT;
 END_STRUCT;
 buffer_UDP_CTT :  STRUCT
  use_long_id : USINT;
  UDP_OK : USINT;
  Customer : ARRAY[0..14] OF UINT;
  Category : ARRAY[0..14] OF UINT;
  Cat : ARRAY[0..4] OF UINT;
  Wgt : ARRAY[0..4] OF USINT;
  BackColor : USINT;
  ForeColor : USINT;
  Future : ARRAY[0..4] OF USINT;
 END_STRUCT;
END_TYPE
```

### Program Logical/Sequences/200ms/USB_Pmem (IEC, version 3.00.0)
